		0://等待激活
			IF   xcmd THEN
			 		xQBusy:=TRUE;
					xQDone:=FALSE;
					iCmdStep :=iCmdStep +1;
					xcmd:=FALSE;
			END_IF
		1://指令
				iCmdStep :=iCmdStep +1;
				iCmdOldStep:=iCmdStep;
		2://开始执行
				xStart :=TRUE;
				iCmdStep :=iCmdStep +1;
				iCmdOldStep:=iCmdStep;
		3://等待接受
					IF   xBusy THEN
					 		iCmdStep :=iCmdStep +1;
					END_IF
					iCmdOldStep:=iCmdStep;
		4://报警待整理数据
				IF  iOperType<> 14  AND  NOT xBusy AND xDone THEN
						iCmdStep :=iCmdStep +1;
				ELSIF iOperType =14 AND  NOT xQNoRead THEN
				 		iCmdStep :=iCmdStep +1;	
				END_IF
				iCmdOldStep:=iCmdStep;
		5://处理接收的数据
					IF iOperType =1 THEN
							IF FIND(strQBarCode,'$R') <> 0 AND FIND(strQBarCode,'I4') <> 0	THEN					
									 CutStrToSeperator('"',strQBarCode);
									 stParOut.sSrialNumber := CutStrToSeperator('"',strQBarCode);
									 iCmdStep :=iCmdStep +1;;	
							END_IF
					ELSIF iOperType =2 THEN
					 					IF FIND(strQBarCode,'$R') <> 0 		THEN
															IF FIND(strQBarCode,'S') <> 0 THEN
																			_Stemp[1]:=RIGHT(strQBarCode,LEN(strQBarCode)-4);
																			_Stemp[2]:=LEFT(_Stemp[1],FIND(_Stemp[1],'g$R')-1);
																			stParOut.rCurrentTareWight := TO_REAL(_Stemp[2]);
																			iCmdStep :=iCmdStep +1;	
															ELSIF FIND(strQBarCode,'T +') <> 0 THEN	
																			eErrorID:=MT_MCK_ERROR.FLT_ZOverMax;
															ELSIF FIND(strQBarCode,'T -') <> 0 THEN	
																			eErrorID:=MT_MCK_ERROR.FLT_ZOverMax;
															ELSIF FIND(strQBarCode,'T I') <> 0 THEN
															 				eErrorID:=MT_MCK_ERROR.FLT_CannotExecutable;			
															END_IF										
									END_IF						
					ELSIF iOperType =3 THEN
					 						IF FIND(strQBarCode,'$R') <> 0 		THEN
															IF FIND(strQBarCode,'TI S') <> 0 OR FIND(strQBarCode,'TI D') <> 0 THEN
																_Stemp[1]:=RIGHT(strQBarCode,LEN(strQBarCode)-4);
																_Stemp[2]:=LEFT(_Stemp[1],FIND(_Stemp[1],'g$R')-1);
																stParOut.rCurrentTareWight := TO_REAL(_Stemp[2]);
																iCmdStep :=iCmdStep +1;;	
															ELSIF FIND(strQBarCode,'TI +') <> 0 THEN	
																eErrorID:=MT_MCK_ERROR.FLT_ZOverMax;
															ELSIF FIND(strQBarCode,'TI -') <> 0 THEN	
																eErrorID:=MT_MCK_ERROR.FLT_ZOverMax;
															ELSIF FIND(strQBarCode,'TI I') <> 0 THEN
															  eErrorID:=MT_MCK_ERROR.FLT_CannotExecutable;			
															END_IF										
												END_IF		
					ELSIF iOperType =4 THEN									
										IF FIND(strQBarCode,'$R') <> 0 AND FIND(strQBarCode,'TA') <> 0	THEN
											 _Stemp[1]:=RIGHT(strQBarCode,LEN(strQBarCode)-5);
											 _Stemp[2]:=LEFT(_Stemp[1],FIND(_Stemp[1],'g$R')-1);
											 stParOut.rCurrentTareWight := TO_REAL(_Stemp[2]);
											 iCmdStep :=iCmdStep +1;;	
										END_IF		
					ELSIF	iOperType =5 THEN		
										IF FIND(strQBarCode,'$R') <> 0 AND FIND(strQBarCode,'TAC') <> 0	THEN
											 stParOut.rCurrentTareWight:=0;
											 iCmdStep :=iCmdStep +1;;	
										 ELSIF FIND(strQBarCode,'EL') <>0 THEN
											 eErrorID:=MT_MCK_ERROR.FLT_LogicaL;//逻辑错误
										 ELSIF FIND(strQBarCode,'ES') <>0 THEN
											 eErrorID:=MT_MCK_ERROR.FLT_Syntax;//语法错误
										 ELSIF FIND(strQBarCode,'I') <>0 THEN
											 eErrorID:=MT_MCK_ERROR.FLT_CommandCantSend;//指令条件不满足,无法发送	
										 ELSIF FIND(strQBarCode,'L') <>0 THEN
											 eErrorID:=MT_MCK_ERROR.FLT_PARA;//参数错误		
										 ELSIF FIND(strQBarCode,'TAC I') <>0 THEN
											 eErrorID:=MT_MCK_ERROR.FLT_CommandCantSend;
										 END_IF																	
					ELSIF  	iOperType =6 THEN													
											IF FIND(strQBarCode,'Z A') <> 0 THEN
													stParOut.rCurrentTareWight :=0;
													stParOut.rCurrentWeight :=0;
													iCmdStep :=iCmdStep +1;;	
											ELSIF FIND(strQBarCode,'Z +') <> 0 THEN
												eErrorID:=MT_MCK_ERROR.FLT_ZOverMax;							
											ELSIF FIND(strQBarCode,'Z -') <> 0 THEN
												eErrorID:=MT_MCK_ERROR.FLT_ZOverMin;				
											ELSIF FIND(strQBarCode,'Z I') <> 0 THEN
												eErrorID:=MT_MCK_ERROR.FLT_CannotExecutable;					
											END_IF			
				ELSIF  	iOperType =7 THEN													
											IF FIND(strQBarCode,'$R') <> 0 	THEN
														 IF FIND(strQBarCode,'ZI') <> 0 AND (FIND(strQBarCode,'S') <> 0 OR FIND(strQBarCode,'D') <> 0) THEN
															 stParOut.rCurrentTareWight :=0;
															 stParOut.rCurrentWeight :=0;
															 iCmdStep :=iCmdStep +1;;	
															ELSIF FIND(strQBarCode,'Z +') <> 0 THEN
																	 eErrorID:=MT_MCK_ERROR.FLT_ZOverMax;							
															 ELSIF FIND(strQBarCode,'Z -') <> 0 THEN
																	 eErrorID:=MT_MCK_ERROR.FLT_ZOverMin;				
																ELSIF FIND(strQBarCode,'Z I') <> 0 THEN
																	 eErrorID:=MT_MCK_ERROR.FLT_ZI;		
																ELSIF	 FIND(strQBarCode,'ZI I') <> 0 THEN
																 	 eErrorID:=MT_MCK_ERROR.FLT_CannotExecutable;
																END_IF
													END_IF
					ELSIF  	iOperType =8 THEN												
											IF FIND(strQBarCode,'$R') <> 0 AND FIND(strQBarCode,'S') <>0		THEN
														IF FIND(strQBarCode,'mg') <> 0 THEN
															_Stemp[1]:=RIGHT(strQBarCode,LEN(strQBarCode)-5);
															_Stemp[2]:=LEFT(_Stemp[1],FIND(_Stemp[1],'g$R')-1);
															stParOut.rCurrentWeight := TO_REAL(_Stemp[2]);
															stParOut.sWeightUnit:='mg';
															iCmdStep :=iCmdStep +1;;	
														ELSE 
															IF FIND(strQBarCode,'g') <> 0 THEN
																_Stemp[1]:=RIGHT(strQBarCode,LEN(strQBarCode)-5);
																_Stemp[2]:=LEFT(_Stemp[1],FIND(_Stemp[1],'g$R')-1);
																stParOut.rCurrentWeight := TO_REAL(_Stemp[2]);
																stParOut.sWeightUnit:='mg';		
																iCmdStep :=iCmdStep +1;;			
															END_IF				
														END_IF
											ELSIF FIND(strQBarCode,'EL') <>0 THEN
														eErrorID:=MT_MCK_ERROR.FLT_LogicaL;//逻辑错误
											ELSIF FIND(strQBarCode,'ES') <>0 THEN
														eErrorID:=MT_MCK_ERROR.FLT_Syntax;//语法错误		
										ELSIF FIND(strQBarCode,'I') <>0 THEN
														eErrorID:=MT_MCK_ERROR.FLT_CommandCantSend;//指令条件不满足,无法发送		
										ELSIF FIND(strQBarCode,'L') <>0 THEN
														eErrorID:=MT_MCK_ERROR.FLT_PARA;//参数错误	
										ELSIF FIND(strQBarCode,'S I') <>0 THEN
											 eErrorID:=MT_MCK_ERROR.FLT_CannotExecutable;
										END_IF			
					ELSIF  	iOperType =9 THEN							
										IF FIND(strQBarCode,'$R') <> 0 AND FIND(strQBarCode,'S') <>0 THEN
													 IF FIND(strQBarCode,'g') <> 0 THEN
														 _Stemp[1]:=RIGHT(strQBarCode,LEN(strQBarCode)-5);
														 _Stemp[2]:=LEFT(_Stemp[1],FIND(_Stemp[1],'g$R')-1);
														 stParOut.rCurrentWeight := TO_REAL(_Stemp[2]);
														 stParOut.sWeightUnit:='mg';	
															iCmdStep :=iCmdStep +1;;				
													 ELSE 
														 IF FIND(strQBarCode,'g') <> 0 THEN
															 _Stemp[1]:=RIGHT(strQBarCode,LEN(strQBarCode)-5);
															 _Stemp[2]:=LEFT(_Stemp[1],FIND(_Stemp[1],'g$R')-1);
															 stParOut.rCurrentWeight := TO_REAL(_Stemp[2]);
															 stParOut.sWeightUnit:='mg';		
																iCmdStep :=iCmdStep +1;;			
														 END_IF				
													 END_IF
													 IF stParOut.rCurrentWeight>stParOut.rWeightMax THEN
														 stParOut.rWeightMax:=stParOut.rCurrentWeight;
													 END_IF
													 IF stParOut.rCurrentWeight<stParOut.rWeightMin THEN
														 stParOut.rWeightMin:=stParOut.rCurrentWeight;
													 END_IF	
													
										ELSIF FIND(strQBarCode,'EL') <>0 THEN
													 eErrorID:=MT_MCK_ERROR.FLT_LogicaL;//逻辑错误
													
										ELSIF FIND(strQBarCode,'ES') <>0 THEN
													 eErrorID:=MT_MCK_ERROR.FLT_Syntax;//语法错误
																
										 ELSIF FIND(strQBarCode,'I') <>0 THEN
													 eErrorID:=MT_MCK_ERROR.FLT_CommandCantSend;//指令条件不满足,无法发送
																	
										ELSIF FIND(strQBarCode,'L') <>0 THEN
													 eErrorID:=MT_MCK_ERROR.FLT_PARA;//参数错误
										ELSIF FIND(strQBarCode,'SI I') <>0 THEN
											 eErrorID:=MT_MCK_ERROR.FLT_CannotExecutable;//无法执行		
										END_IF		
				ELSIF  	iOperType =10 THEN										
												IF FIND(strQBarCode,'$R') <> 0 AND FIND(strQBarCode,'S') <>0				THEN
													 IF FIND(strQBarCode,'g') <> 0 THEN
														 _Stemp[1]:=RIGHT(strQBarCode,LEN(strQBarCode)-5);
														 _Stemp[2]:=LEFT(_Stemp[1],FIND(_Stemp[1],'g$R')-1);
														 stParOut.rCurrentWeight := TO_REAL(_Stemp[2]);
														 stParOut.sWeightUnit:='mg';
														 iCmdStep :=iCmdStep +1;;	
													 ELSE 
														 IF FIND(strQBarCode,'g') <> 0 THEN
															 _Stemp[1]:=RIGHT(strQBarCode,LEN(strQBarCode)-5);
															 _Stemp[2]:=LEFT(_Stemp[1],FIND(_Stemp[1],'g$R')-1);
															 stParOut.rCurrentWeight := TO_REAL(_Stemp[2]);
															 stParOut.sWeightUnit:='mg';	
																iCmdStep :=iCmdStep +1;;				
														 END_IF				
													 END_IF
										 ELSIF FIND(strQBarCode,'EL') <>0 THEN
											 eErrorID:=MT_MCK_ERROR.FLT_LogicaL;//逻辑错误
										 ELSIF FIND(strQBarCode,'ES') <>0 THEN
											 eErrorID:=MT_MCK_ERROR.FLT_Syntax;//语法错误				
										 ELSIF FIND(strQBarCode,'I') <>0 THEN
											 eErrorID:=MT_MCK_ERROR.FLT_CommandCantSend;//指令条件不满足,无法发送 			
										 ELSIF FIND(strQBarCode,'L') <>0 THEN
											 eErrorID:=MT_MCK_ERROR.FLT_PARA;//参数错误
										 ELSIF FIND(strQBarCode,'SIR I') <>0 THEN
											 eErrorID:=MT_MCK_ERROR.FLT_CannotExecutable;//无法执行
										END_IF
				ELSIF  	iOperType =11 THEN										 
									IF FIND(strQBarCode,'$R') <> 0 AND FIND(strQBarCode,'S') <> 0		THEN
												 _Stemp[1]:=RIGHT(strQBarCode,LEN(strQBarCode)-4);
											_Stemp[2]:=LEFT(_Stemp[1],FIND(_Stemp[1],'g$R')-1);
											stParOut.rCurrentWeight := TO_REAL(_Stemp[2]);
											iCmdStep :=iCmdStep +1;;	
									END_IF														 
				ELSIF  	iOperType =12 THEN						
					 				IF FIND(strQBarCode,'$R') <> 0 AND FIND(strQBarCode,'I4') <> 0	THEN
										CutStrToSeperator('"',strQBarCode);
										stParOut.sSrialNumber := CutStrToSeperator('"',strQBarCode);
										iCmdStep :=iCmdStep +1;	
									END_IF
				ELSIF  	iOperType =13 THEN			
								IF FIND(strQBarCode,'$R') <> 0 AND FIND(strQBarCode,'I4') <> 0	THEN
												iCmdStep :=iCmdStep +1;	
								ELSE			
								 					iCmdStep :=2;	
								END_IF
				ELSIF   iOperType =14 THEN	
							  IF FIND(strQBarCode,'$R') <> 0 AND FIND(strQBarCode,'S S') <> 0	THEN
									//稳态
								 				IF    FIND(strQBarCode,'g')<>0 THEN
												   // stParOut.rRepeatWeight:=strQBarCode;
													//	stParOut.rStableWeight:=strQBarCode;
													_Stemp[1]:=RIGHT(strQBarCode,LEN(strQBarCode)-5);
													_Stemp[2]:=LEFT(_Stemp[1],FIND(_Stemp[1],'g$R')-1);
													stParOut.rRepeatWeight:=TO_REAL(_Stemp[2]);
													stParOut.rStableWeight:=stParOut.rRepeatWeight;
													xRepeatReceive:=TRUE;;
												ELSE
												 			eErrorID:=MT_MCK_ERROR.FLT_SIRERROR;
												 END_IF
												iCmdStep :=iCmdStep +1;	
								ELSIF  	FIND(strQBarCode,'$R') <> 0 AND FIND(strQBarCode,'S D')<>0 THEN
								 //非稳态
								 					IF    FIND(strQBarCode,'g')<>0 THEN
																_Stemp[1]:=RIGHT(strQBarCode,LEN(strQBarCode)-5);
																_Stemp[2]:=LEFT(_Stemp[1],FIND(_Stemp[1],'g$R')-1);
																stParOut.rRepeatWeight:=TO_REAL(_Stemp[2]);
													 			xRepeatReceive:=TRUE;
													ELSE
												 			eErrorID:=MT_MCK_ERROR.FLT_SIRERROR;
												 END_IF
												iCmdStep :=iCmdStep +1;	
								ELSIF  FIND(strQBarCode,'S I')<>0 THEN
								 			eErrorID:=MT_MCK_ERROR.FLT_CannotExecutable;//无法执行
								ELSIF  FIND(strQBarCode,'S L')<>0 THEN
								 			eErrorID:=MT_MCK_ERROR.FLT_PARA;//参数错误
								ELSIF  FIND(strQBarCode,'S +')<>0 THEN
								 			eErrorID:=MT_MCK_ERROR.FLT_SIROverMax;
								ELSIF  FIND(strQBarCode,'S -')<>0 THEN
								 			eErrorID:=MT_MCK_ERROR.FLT_SIROverMIN;
								END_IF				
				END_IF
				iCmdOldStep:=iCmdStep;
		6:	
						xQDone:=TRUE;
						xQBusy:=FALSE;	
						iCmdOldStep:=iCmdStep;
						iCmdStep :=0;		
	END_CASE
END_ACTION

ACTION ACT_Error:
IF  eErrorID <> 0 THEN
	xQError:=TRUE;
END_IF
//报错内容输出
CASE eErrorID OF 
	MT_MCK_ERROR.FLT_CMD_TIMEOUT:
		stParOut.sErrorID:='FLT_CMD_TIMEOUT';
	MT_MCK_ERROR.FLT_CmdFeedback:
		stParOut.sErrorID:='FLT_CmdFeedback';
	MT_MCK_ERROR.FLT_CommandCantSend:
		stParOut.sErrorID:='FLT_CommandCantSend';
	MT_MCK_ERROR.FLT_CONNECT:
		stParOut.sErrorID:='FLT_CONNECT';
	MT_MCK_ERROR.FLT_LogicaL:
		stParOut.sErrorID:='FLT_LogicaL';
	MT_MCK_ERROR.FLT_Par:
		stParOut.sErrorID:='FLT_Par';
	MT_MCK_ERROR.FLT_PARA:
		stParOut.sErrorID:='FLT_PARA';
	MT_MCK_ERROR.FLT_RDYCMD:
		stParOut.sErrorID:='FLT_RDYCMD';
	MT_MCK_ERROR.FLT_STOP_TIMEOUT:
		stParOut.sErrorID:='FLT_STOP_TIMEOUT';
	MT_MCK_ERROR.FLT_Syntax:
		stParOut.sErrorID:='FLT_Syntax';
	MT_MCK_ERROR.FLT_TOverMax:
		stParOut.sErrorID:='FLT_TOverMax';
	MT_MCK_ERROR.FLT_TOverMin:
		stParOut.sErrorID:='FLT_TOverMin';
	MT_MCK_ERROR.FLT_ZI:
		stParOut.sErrorID:='FLT_ZI';
	MT_MCK_ERROR.FLT_ZOverMax:
		stParOut.sErrorID:='FLT_ZOverMax';
	MT_MCK_ERROR.FLT_ZOverMin:
		stParOut.sErrorID:='FLT_ZOverMin';
	MT_MCK_ERROR.FLT_CannotExecutable:
			stParOut.sErrorID:='FLT_CannotExecutable';	
	MT_MCK_ERROR.No_ERROR:
		stParOut.sErrorID:='No_ERROR';		
END_CASE
END_ACTION

ACTION ACT_OP:
OperR_TRIG[1](CLK:= (xManualMode AND  stDeviceOpe.xReadSerialNum_HMI) OR((xAutoMode OR  xIDeviceRunning) AND stDeviceOpe.xReadSerialNum_Auto) , Q=> );	//获取序列号,I4			
OperR_TRIG[2](CLK:= (xManualMode AND  stDeviceOpe.xShelling_HMI) OR((xAutoMode OR  xIDeviceRunning) AND stDeviceOpe.xShelling_Auto) , Q=> );		//稳态去皮重,T		
OperR_TRIG[3](CLK:= (xManualMode AND  stDeviceOpe.xShellingInstanly_HMI) OR((xAutoMode OR  xIDeviceRunning) AND stDeviceOpe.xShellingInstanly_HMI) , Q=> );	//立即去皮重,TI			
OperR_TRIG[4](CLK:= (xManualMode AND  stDeviceOpe.xSetTare_HMI) OR((xAutoMode OR  xIDeviceRunning) AND stDeviceOpe.xSetTare_Auto) , Q=> );		//预置皮重，TA		
OperR_TRIG[5](CLK:= (xManualMode AND  stDeviceOpe.xlearTare_HMI) OR((xAutoMode OR  xIDeviceRunning) AND stDeviceOpe.xlearTare_Auto) , Q=> );	//清除皮重,TAC			
OperR_TRIG[6](CLK:= (xManualMode AND  stDeviceOpe.xClearZero_HMI) OR((xAutoMode OR  xIDeviceRunning) AND stDeviceOpe.xClearZero_Auto) , Q=> );	//稳态清零,Z	
OperR_TRIG[7](CLK:= (xManualMode AND  stDeviceOpe.xClearZeroInstanly_HMI) OR((xAutoMode OR  xIDeviceRunning) AND stDeviceOpe.xClearZeroInstanly_Auto) , Q=> );	////立即清零,ZI	
OperR_TRIG[8](CLK:= (xManualMode AND  stDeviceOpe.xAcquireWeight_Steady_HMI) OR((xAutoMode OR  xIDeviceRunning) AND stDeviceOpe.xClearZero_Auto) , Q=> );	////单次获取稳态重量,S	
OperR_TRIG[9](CLK:= (xManualMode AND  stDeviceOpe.xAcquireWeight_RealTime_HMI) OR((xAutoMode OR  xIDeviceRunning) AND stDeviceOpe.xAcquireWeight_RealTime_Auto) , Q=> );	////连续获取重量,SI
OperR_TRIG[10](CLK:= (xManualMode AND  stDeviceOpe.xAcquireWeight_Continuous_HMI) OR((xAutoMode OR  xIDeviceRunning) AND stDeviceOpe.xAcquireWeight_Continuous_Auto) , Q=> );	////连续获取重量,SIR	
OperR_TRIG[11](CLK:= (xManualMode AND  stDeviceOpe.xAcquireWeight_Stop_HMI) OR((xAutoMode OR  xIDeviceRunning) AND stDeviceOpe.xAcquireWeight_Stop_Auto) , Q=> );	///中断连续获取重量,SI
OperR_TRIG[12](CLK:= (xManualMode AND  stDeviceOpe.xRestart_HMI) OR((xAutoMode OR  xIDeviceRunning) AND stDeviceOpe.xRestart_Auto) , Q=> );	//重启秤体	
OperR_TRIG[13](CLK:=xIReset , Q=> );	//Cancel	
OperR_TRIG[14](CLK:=( (xManualMode AND  stDeviceOpe.xRepeatRead_Hmi ) OR((xAutoMode OR  xIDeviceRunning) AND stDeviceOpe.xRepeatRead_Auto) )AND iOperType <>14 , Q=> );	//循环读取重量并显示
FOR  i:= 1 TO 20 BY 1 DO
 	IF   OperR_TRIG[i].Q THEN
				iOperType:= i;
				xCmd:=TRUE;
				EXIT;
	END_IF
END_FOR

IF   iOperType =1 THEN
 	strRead := 'I4$R$N';
ELSIF   iOperType =2 THEN
 	strRead := 'T$R$N';
ELSIF   iOperType =3 THEN
 	strRead := 'TI$R$N';
ELSIF   iOperType =4 THEN
 	_sSendData := CONCAT(_sSendData,'TA');
	_sSendData := CONCAT(_sSendData,' ');		
	_sSendData := CONCAT(_sSendData,TO_STRING(rTareSet));
	_sSendData := CONCAT(_sSendData,' ');
	_sSendData := CONCAT(_sSendData,'g');//单位
	_sSendData := CONCAT(_sSendData,'$R$N');//回车换行符			
 	strRead := _sSendData;
ELSIF   iOperType =5 THEN
 	strRead := 'TAC$R$N';
ELSIF   iOperType =6 THEN
 	strRead := 'Z$R$N';
ELSIF   iOperType =7 THEN
 	strRead := 'ZI$R$N';
ELSIF   iOperType =8 THEN
 	strRead := 'S$R$N';
ELSIF   iOperType =9 THEN
 	strRead := 'SI$R$N';
ELSIF   iOperType =10 THEN
 	strRead := 'SIR$R$N';
ELSIF   iOperType =11 THEN
 	strRead := 'SI$R$N';
ELSIF   iOperType =12 THEN
 	strRead := 'R01$R$N';
ELSIF iOperType =13 THEN
 	strRead := '@$R$N';
ELSIF  iOperType =14 THEN
  strRead := 'SIR$R$N';
END_IF

	stDeviceOpe.xReadSerialNum_HMI:=stDeviceOpe.xReadSerialNum_Auto :=FALSE;	//获取序列号,I4
	stDeviceOpe.xShelling_HMI:=stDeviceOpe.xShelling_Auto						:=FALSE;//稳态去皮重,T
	stDeviceOpe.xShellingInstanly_HMI:=stDeviceOpe.xShellingInstanly_Auto	:=FALSE;//立即去皮重,TI	
	stDeviceOpe.xSetTare_HMI:=stDeviceOpe.xSetTare_Auto										:=FALSE;//预置皮重，TA
	stDeviceOpe.xlearTare_HMI:=stDeviceOpe.xlearTare_Auto									:=FALSE;//清除皮重,TAC
	stDeviceOpe.xClearZero_HMI:=stDeviceOpe.xClearZero_Auto								:=FALSE;//稳态清零,Z
	stDeviceOpe.xClearZeroInstanly_HMI:=stDeviceOpe.xClearZeroInstanly_Auto:=FALSE;//立即清零,ZI
	stDeviceOpe.xAcquireWeight_Steady_HMI:=stDeviceOpe.xAcquireWeight_Steady_Auto :=FALSE;//单次获取稳态重量,S
	stDeviceOpe.xAcquireWeight_RealTime_HMI:=stDeviceOpe.xAcquireWeight_RealTime_Auto:=FALSE;//连续获取重量,SI
	stDeviceOpe.xAcquireWeight_Continuous_HMI:=stDeviceOpe.xAcquireWeight_Continuous_Auto:=FALSE;//连续获取重量,SIR
	stDeviceOpe.xAcquireWeight_Stop_HMI:=stDeviceOpe.xAcquireWeight_Stop_Auto		:=FALSE;//中断连续获取重量,SI
	stDeviceOpe.xRestart_HMI:=stDeviceOpe.xRestart_Auto										      :=FALSE;//重启秤体	
	stDeviceOpe.xRepeatRead_Hmi:=stDeviceOpe.xRepeatRead_Auto							      :=FALSE;//重复读取
	//xIReset:=FALSE;
END_ACTION

ACTION ACT_Reset:
IF ( xIReset = TRUE )THEN
 		iCmdStep:=0;
  	iStep := 0 ;
		iLoadStep:=0;
  	xQError := FALSE ;
  	xBusy  := FALSE;
		xQBusy  := FALSE;
		xStart  := FALSE;
		eErrorID:=MT_MCK_ERROR.No_ERROR;
		iCmdOldStep:=0;
		xIReset:=FALSE;
END_IF
END_ACTION

ACTION ACT_RW:

 
IF ( First = FALSE )THEN
   	TcpIpClient.sRemoteServer := stSysPar.sRemoteHost;
 		TcpIpClient.nRemotePort := stSysPar.nRemotePort;
   	TcpIpClient.pSendData := ADR(ClientSendBuffer);
   	TcpIpClient.pRecvData := ADR(ClientRecvBuffer);
   	First := TRUE ;
ELSE
  	TcpIpClient(iStep :=	eStepCmd );
 	CASE iStep OF
		0: (* wait start *)
		   	IF ( xStart = FALSE )THEN
		       	xDone := FALSE ;
		   	END_IF
		  	IF ( xStart = FALSE ) AND( xDone = FALSE )THEN
		       	xRdyCmd := TRUE  ;
		   	END_IF

		   	IF ( xStart = TRUE ) AND( xRdyCmd = TRUE )THEN
				iStep  :=  10 ;
				xBusy:=TRUE;
			  xRdyCmd := FALSE  ;
			(*ELSE
 			 	xBusy  := FALSE;*)
		   	END_IF

		10: (* creat soket*)
			xStart := FALSE;
			MEMSET(ADR(strLocalQBarCode),0,SIZEOF(strLocalQBarCode));
			MEMSET(ADR(strQBarCode),0,SIZEOF(strQBarCode));
			MEMSET(ADR(ClientRecvBuffer),0,SIZEOF(ClientRecvBuffer));
			eStepCmd := CLIENT_STATE_CONNECT_START ;
		    	iStep := 20 ;

		20: (* socket ok *)
 			 IF( eStepCmd = CLIENT_STATE_IDLE )THEN
		    	 	iStep := 30 ;
			ELSIF( eStepCmd = CLIENT_STATE_ERROR )THEN
				iQErrorNo:=iStep;
		    	 	iStep := 100 ;
	         	END_IF

		30: (* send read *)
   			MEMCPY(ADR(ClientSendBuffer),ADR(strRead),SIZEOF(strRead));
			TcpIpClient.SendLen := LEN(strRead);
			eStepCmd := CLIENT_STATE_SEND_START ;
		    	iStep := 40 ;

		40: (* send ok *)
 			IF( eStepCmd = CLIENT_STATE_IDLE )THEN
		    	 	iStep := 50 ;
			ELSIF( eStepCmd = CLIENT_STATE_ERROR )THEN
				iQErrorNo:=iStep;
		    	 	iStep := 999 ;
	         	END_IF

		50: (* recive read *)
			xQNoRead:=TRUE;
			eStepCmd := CLIENT_STATE_RECIVE_START ;
		    	iStep := 55 ;

   55:
			strLocalQBarCode:='';
			strQBarCode:='';
			Waittime(IN:=TRUE, PT:= t#20ms);
	      	IF(waittime.Q = TRUE )THEN
 							Waittime(IN:= FALSE);
		    	 		iStep := 60 ;
	        END_IF

		60: (* recive end *)
				IF( eStepCmd = CLIENT_STATE_IDLE )THEN
						 MEMCPY(ADR(strLocalQBarCode),ADR(ClientRecvBuffer),TcpIpClient.cbReceived);
						 strQBarCode:=MID(strLocalQBarCode,iICodeLEN,iICodePOS);
						 iStep := 80 ;
			 ELSIF( eStepCmd = CLIENT_STATE_ERROR )THEN
				 		 iQErrorNo:=iStep;
						 iStep := 70;
			 END_IF
		70:
				MEMSET(ADR(strLocalQBarCode),0,SIZEOF(strLocalQBarCode));
				MEMSET(ADR(strQBarCode),0,SIZEOF(strQBarCode));
				iStep := 80;

		80: (* close socket *)
			 IF  strQBarCode<>'' THEN
							 xQNoRead:=FALSE;
			 ELSE
							 xQNoRead:=TRUE;
			 END_IF
			 IF iOperType =14 THEN
					 	iStep := 50 ;
			 ELSE
				 		iStep := 100 ;
			 END_IF
		100: (* close socket *)
					eStepCmd := CLIENT_STATE_CLOSE_START ;
		    	iStep := 110 ;
		110: (* recive end *)
				IF( eStepCmd = CLIENT_STATE_IDLE )THEN
							xBusy  := FALSE;
							xDone := TRUE ;
							iStep := 0 ;
				ELSIF( eStepCmd = CLIENT_STATE_ERROR )THEN
							iStep := 999 ;
							END_IF

		999: (* Done *)
				 xBusy:=FALSE;
				 xQError := TRUE ;
					iStep := 0 ;
	END_CASE
END_IF
END_ACTION

END_FUNCTION_BLOCK

// ---- POUs/003_FB/0008_LocalClient/FB_LocalClient.TcPOU
FUNCTION_BLOCK FB_LocalClient
VAR_INPUT
	sRemoteServer		: STRING(15) := '192.168.0.3';(* IP adress of remote server *)
	nRemotePort			: UDINT := 1030;
    RecvTime            : TIME ;
	pSendData           : POINTER TO BYTE ;
    SendLen             : INT ;
	pRecvData           : POINTER TO BYTE ;
    RecvLen             : INT := 255 ;


    Start             : BOOL ;
    Send              : BOOL ;
    Recv              : BOOL ;
    Close             : BOOL ;

END_VAR
VAR_OUTPUT
			hSocket				: T_HSOCKET;
			bBusy 				: BOOL;
			bError				: BOOL;
			nErrId				: UDINT;
    Connected           : BOOL ;
    SendOK              : BOOL ;
    RecvOK              : BOOL ;
    Closed              : BOOL ;
    RdyCmd              : BOOL ;
	Done: BOOL;
END_VAR

VAR_IN_OUT
    iStep             : E_ClientSteps;
END_VAR


VAR
	
	
	fbConnect 		: FB_SocketConnect := ( sSrvNetId := ''  );
	fbClose				: FB_SocketClose := ( sSrvNetId := '', tTimeout := DEFAULT_ADS_TIMEOUT );
	fbSocketSend		: FB_SocketSend      := ( sSrvNetID := '', tTimeout := DEFAULT_ADS_TIMEOUT );
	fbSocketReceive        : FB_SocketReceive := ( sSrvNetID := '', tTimeout := DEFAULT_ADS_TIMEOUT );
	fbConnectTON		: TON := ( PT := PLCPRJ_RECONNECT_TIME );
	fbDataExchaTON		: TON := ( PT := PLCPRJ_SEND_CYCLE_TIME );
	fbReceiveTON		: TON;
	fbDisconnectTON      : TON;
    arrayRecive                 : ARRAY [1..1000] OF BYTE ;
	a,b,c,d : BOOL ;

	cbReceived, startPos, endPos, idx	: UDINT;
	cbFrame				: UDINT;
	rxBuffer				: ARRAY[0..MAX_PLCPRJ_RXBUFFER_SIZE] OF BYTE;
	
END_VAR

CASE iStep OF
	CLIENT_STATE_IDLE:
	;
	CLIENT_STATE_CONNECT_START:
		  IF ( Connected =  FALSE )
		  THEN
				fbConnectTON( IN := TRUE, PT := PLCPRJ_RECONNECT_TIME );
						IF fbConnectTON.Q THEN
							fbConnectTON( IN := FALSE );
							fbConnect(  bExecute := FALSE  );
							fbConnect(	sRemoteHost		:= sRemoteServer,
										nRemotePort		:= nRemotePort,
										bExecute		:= TRUE );
							iStep := CLIENT_STATE_CONNECT_WAIT;
						END_IF

	    	ELSE
			   iStep := CLIENT_STATE_IDLE;
			END_IF

   CLIENT_STATE_CONNECT_WAIT:
				fbConnect( bExecute := FALSE );
				IF NOT fbConnect.bBusy THEN
					IF NOT fbConnect.bError THEN
						Connected 	:= TRUE;
						hSocket 	:= fbConnect.hSocket;
						iStep := CLIENT_STATE_IDLE;

					ELSE

						nErrId := fbConnect.nErrId;
						iStep := CLIENT_STATE_ERROR;
					END_IF
				END_IF


	CLIENT_STATE_SEND_START:
		fbSocketSend( bExecute := FALSE );
		fbSocketSend( 	hSocket	:= hSocket,
						pSrc	:= pSendData,
						cbLen	:= SendLen,(* string length inclusive zero delimiter *)
						bExecute:= TRUE );
		cbReceived	:= 0 ;
		MEMSET(ADR(rxBuffer),0,SIZEOF(rxBuffer));
		iStep := CLIENT_STATE_SEND_WAIT;

	CLIENT_STATE_SEND_WAIT:
		fbSocketSend( bExecute := FALSE );
		IF NOT fbSocketSend.bBusy THEN
			IF NOT fbSocketSend.bError THEN
				iStep := CLIENT_STATE_IDLE;
			ELSE

				nErrId := fbSocketSend.nErrId;
				iStep := CLIENT_STATE_CLOSE_START;
			END_IF
		END_IF
	CLIENT_STATE_WAITTIME1:
		iStep := CLIENT_STATE_WAITTIME2;
	CLIENT_STATE_WAITTIME2:
		iStep := CLIENT_STATE_RECIVE_START;

	CLIENT_STATE_RECIVE_START:
		fbDisconnectTON(  );
		fbReceiveTON( IN := TRUE );
		IF fbReceiveTON.Q THEN
			fbReceiveTON( IN := FALSE );
			fbSocketReceive( bExecute := FALSE );
			fbSocketReceive(  hSocket:= hSocket,
							pDest:= ADR( rxBuffer ) + cbReceived,
							cbLen:= SIZEOF( rxBuffer ) - cbReceived,
							bExecute:= TRUE );
			iStep := CLIENT_STATE_RECIVE_WAIT;
		END_IF

	CLIENT_STATE_RECIVE_WAIT:
		fbSocketReceive( bExecute := FALSE );
		IF NOT fbSocketReceive.bBusy THEN
			IF NOT fbSocketReceive.bError THEN

				IF (fbSocketReceive.nRecBytes > 0) THEN(* bytes received *)

					startPos 		:= cbReceived;(* rxBuffer array index of first data byte *)
					endPos  		:= cbReceived + fbSocketReceive.nRecBytes  - 1;(* rxBuffer array index of last data byte *)
					cbReceived 	:= cbReceived + fbSocketReceive.nRecBytes;(* calculate the number of received data bytes *)
					cbFrame		:= 0;(* reset frame length *)

					IF cbReceived < RecvLen THEN(* no overflow *)

						fbReceiveTON( PT := T#0s ); (* bytes received => increase the read (polling) speed *)
						fbDisconnectTON( IN := FALSE );(* bytes received => disable timeout check *)

						(* search for string end delimiter *)
						FOR idx := startPos TO endPos BY 1 DO
							IF rxBuffer[idx] = 0 THEN(* string end delimiter found *)
								cbFrame := idx + 1;(* calculate the length of the received string (inclusive the end delimiter) *)
								MEMCPY(  pRecvData, ADR( rxBuffer ), cbFrame );(* copy the received string to the output variable (inclusive the end delimiter) *)
								MEMMOVE( ADR( rxBuffer ), ADR( rxBuffer[cbFrame] ),  cbReceived - cbFrame  );(* move the reamaining data bytes *)
								cbReceived := cbReceived - cbFrame;(* recalculate the reamaining data byte length *)
								a := TRUE ;
								iStep := CLIENT_STATE_IDLE;
								EXIT;
							END_IF
						END_FOR

					ELSE(* there is no more free read buffer space => the answer string should be terminated *)
						b := TRUE ;
						nErrId := PLCPRJ_ERROR_RECEIVE_BUFFER_OVERFLOW;(* buffer overflow !*)
						iStep := CLIENT_STATE_CLOSE_START;
					END_IF

				ELSE(* no bytes received *)
					fbReceiveTON( PT := PLCPRJ_RECEIVE_POLLING_TIME );(* no bytes received => decrease the read (polling) speed *)
					fbDisconnectTON( IN := TRUE, PT := PLCPRJ_RECEIVE_TIMEOUT );(* no bytes received => enable timeout check*)
					IF fbDisconnectTON.Q THEN (* timeout error*)
						fbDisconnectTON( IN := FALSE );
						c := TRUE ;
						nErrID := PLCPRJ_ERROR_RECEIVE_TIMEOUT;
						iStep := CLIENT_STATE_IDLE;
					ELSE(* repeat reading *)
						iStep := CLIENT_STATE_RECIVE_START; (* repeat reading *)
					END_IF
				END_IF
			ELSE(* receive error *)
				d := TRUE ;
				nErrId := fbSocketReceive.nErrId;
				iStep := CLIENT_STATE_CLOSE_START;
			END_IF
		END_IF



	CLIENT_STATE_CLOSE_START:
	    fbClose( bExecute := FALSE );
		fbClose(	hSocket:= hSocket,
				bExecute:= TRUE );
		iStep := CLIENT_STATE_CLOSE_WAIT;

	CLIENT_STATE_CLOSE_WAIT:
		fbClose( bExecute := FALSE );
		IF NOT fbClose.bBusy THEN

			Connected := FALSE;
			MEMSET( ADR(hSocket), 0, SIZEOF(hSocket));
			IF fbClose.bError THEN

				nErrId := fbClose.nErrId;
				iStep := CLIENT_STATE_ERROR;
			ELSE
				bBusy := FALSE;
				bError := FALSE;
				nErrId := 0;
				iStep := CLIENT_STATE_IDLE;
			END_IF
		END_IF

	CLIENT_STATE_ERROR:
		bError := TRUE;
		IF Connected THEN
			iStep := CLIENT_STATE_CLOSE_START;
		ELSE
			bBusy := FALSE;
			(* iStep := CLIENT_STATE_IDLE *);
		END_IF

END_CASE

END_FUNCTION_BLOCK

// ---- POUs/003_FB/0007_Vacuum/FB_SmcVacuum.TcPOU
FUNCTION_BLOCK FB_SmcVacuum
(*
********************************************************************************
* Name: FB_Encoder
*
* Author:  AutomanH
* Version: 1.0.0
*
* Description:
*   
* Remarks:
*
* Revisions:
* V1.0.0-Automanh Build
* 
*********************************************************************************)
VAR_INPUT
 xIAutoMode:BOOL;
 xIManualMode:BOOL;
 xIVacuumWork:BOOL;//供给阀工作
 xIVacuumBroken:BOOL;//破坏阀工作
 xIVacuumWorkHMI:BOOL;
 xIVacuumBrokenHMI:BOOL;
 xIDeviceRunning:BOOL;
 xIVacuumWorkReached:BOOL;//真空度达到
 xIVacuumBrokenReached:BOOL;//真空以破坏
END_VAR
VAR_OUTPUT
 xQVacuumFeedValve:BOOL;//供给阀输出
 xQVacuumBrokenValve:BOOL;//破坏阀输出
END_VAR

VAR
 VacuumR_TRIG	:	R_TRIG;
VacuumBrokenR_TRIG:R_TRIG;
END_VAR

VacuumR_TRIG(CLK:= ((xIAutoMode OR xIDeviceRunning)AND xIVacuumWork) OR (xIManualMode	AND xIVacuumWorkHMI) , Q=> );
VacuumBrokenR_TRIG(CLK:= ((xIAutoMode OR xIDeviceRunning )AND  xIVacuumBroken) OR (fbMachine[1].xManualMode AND xIVacuumBrokenHMI) , Q=> );
//真空吸
IF	VacuumR_TRIG.Q THEN 
	xQVacuumFeedValve	:= TRUE ;//	卡片搬运工位¶真空发生器1¶供给阀控制
	xQVacuumBrokenValve:=FALSE;//	卡片搬运工位¶真空发生器1¶破坏阀控制
//	xIVacuumWork:=FALSE;
//	xIVacuumWorkHMI:=FALSE;
END_IF 

//真空吸
IF VacuumBrokenR_TRIG.Q THEN 
	xQVacuumBrokenValve	:= TRUE ;
	xQVacuumFeedValve:=FALSE;
//	xIVacuumBroken:=FALSE;
//	xIVacuumBrokenHMI:=FALSE;
END_IF 
IF			xQVacuumBrokenValve AND  xIVacuumBrokenReached THEN
 				xQVacuumBrokenValve	:= FALSE ;
END_IF

	xIVacuumWork:=FALSE;
	xIVacuumWorkHMI:=FALSE;
	xIVacuumBroken:=FALSE;
	xIVacuumBrokenHMI:=FALSE;

END_FUNCTION_BLOCK

// ---- POUs/003_FB/0010_LoadCell/FB_LoadCell.TcPOU
FUNCTION_BLOCK FB_LoadCell EXTENDS FB_Modbus_Tcp
(*
********************************************************************************
* Name: FB_LoadCell
*
* Author:  Automanh
* Version: 1.0.0
*
* Description:
*  LoadSell of XJC-CF3600-F
*
* Remarks:
*
* Revisions:
*   1.0 -AutomanH Rebuild
*********************************************************************************)
VAR_INPUT
xIStart:BOOL;
xIReset:BOOL;
LocalClient:stModbusPara;
stDeviceOpe	:DUT_DeviceOpe;
xIDeviceRunning:BOOL;
xManualMode:BOOL;
xAutoMode:BOOL;
END_VAR
VAR_OUTPUT
 xQRdyCmd:BOOL;
 xQBusy:BOOL;
 xQError:BOOL;
 xQDone:BOOL;
 xQZeroSingle:BOOL;
 stParOut	: ST_LoadCell_ParOut;//参数输出
END_VAR
VAR
	// modbustcp连接步骤
	iCmdStep,iCmdOldStep: INT;
	wLEN:INT;
	wADDR:INT;
	strFunCode:STRING; 
	
	OperR_TRIG:ARRAY[1..20] OF R_TRIG;
	tTimeout:TON;
	tonDelay:TON;
	eErrorID		: ST_LoadCell_Error;(*错误码*)
	// 操作类型
	iOperType: INT;
	i:INT;
	rTempData:REAL;
END_VAR

MEMCPY(ADR(SUPER^.stModbusPara),ADR(LocalClient),SIZEOF(localClient));
SUPER^.M_Modbus();
ACT_Op();
ACT_Cmd();
ACT_Reset();
ACT_Error();

ACTION ACT_Cmd:

IF  NOT  xQBusy THEN
 		xQRdyCmd:=TRUE;
ELSE
 		xQRdyCmd:=FALSE;	
END_IF
tTimeout(IN:= iCmdStep =iCmdOldStep AND iCmdStep<>0 , PT:= T#5S, Q=> , ET=> );
IF		tTimeout.Q THEN
 	xQError:=TRUE;
	eErrorID:=ST_LoadCell_Error.FLT_CMD_TIMEOUT;
END_IF
	 
CASE iCmdStep OF
		0: //等待启动
			 	IF  xIStart THEN
					xQBusy:=TRUE;
					xQDone:=FALSE;
					xIStart:=FALSE;
					iCmdStep:=iCmdStep +1;
				END_IF
		1://等待选择modbusTcp功能码
			 		iCmdOldStep:=iCmdStep;
					iCmdStep:=iCmdStep +1;
		2://判断
					iCmdOldStep:=iCmdStep;
					IF   strFunCode = '10H' THEN
							 tonDelay(IN:= FALSE);
							xQZeroSingle:=TRUE;
							iCmdStep:=iCmdStep +1;
					ELSIF strFunCode = '04H' THEN
					 		iCmdStep:=iCmdStep +2;
					END_IF
					
		3://等待至少20ms以上
				iCmdOldStep:=iCmdStep;
				 tonDelay(IN:= TRUE, PT:=T#100MS , Q=> , ET=> );
				 IF  tonDelay.Q THEN
								 tonDelay(IN:= FALSE);
								xQZeroSingle:=FALSE;
								iCmdStep:=iCmdStep +1;
				 END_IF
		4://读取当前GROSS值
	  					 wQuantityReadInputRegs:=wLEN;(*读取个数*)
	  					 wMBAddReadInputRegs:=wADDR;(*读取起始地址*)
	  					 xReadInputRegs:= TRUE;	
	  				 IF  fbReadInputRegs.bBusy  THEN
	  								xReadInputRegs:=FALSE;
	  							 iCmdOldStep:=iCmdStep;
	  							 iCmdStep:=iCmdStep +1;
	  				 END_IF	
	  5://接收数据
	  	 	iCmdOldStep:=iCmdStep;
	  	 	IF  NOT 	fbReadInputRegs.bBusy AND  NOT  	fbReadInputRegs.bError THEN
				 				MEMCPY(ADR(rTempData),ADR(arwDataReadRegs[1]),SIZEOF(rTempData));
								stParOut.rGROSSWeight:=rTempData;
	  						iCmdStep:=iCmdStep +1;
	  		ELSIF   	fbReadInputRegs.bError THEN
	  					iCmdStep:=0;		
	  					eErrorID:=ST_LoadCell_Error.FLT_PARA;					
	  		END_IF	
		6:
			 		xQDone:=TRUE;
					xQBusy:=FALSE;	 
					iCmdOldStep:=iCmdStep;		
					iCmdStep :=0;					 
END_CASE;
END_ACTION

ACTION ACT_Error:
IF  eErrorID <> 0 THEN
	xQError:=TRUE;
END_IF
//报错内容输出
CASE eErrorID OF 
 	ST_LoadCell_Error.No_ERROR:
		stParOut.sErrorID:='NO ERROR';
	ST_LoadCell_Error.FLT_CMD_TIMEOUT:
		stParOut.sErrorID:='FLT_CMD_TIMEOUT';
	ST_LoadCell_Error.FLT_PARA:
		stParOut.sErrorID:='FLT_PARA';
	
	
END_CASE
END_ACTION

ACTION ACT_OP:
OperR_TRIG[1](CLK:= (xManualMode AND  stDeviceOpe.xReadGROSSHmi) OR((xAutoMode OR  xIDeviceRunning) AND stDeviceOpe.xReadGROSSAuto) , Q=> );	//获取总值GROSS		
OperR_TRIG[2](CLK:= (xManualMode AND  stDeviceOpe.XSetZEROHmi) OR((xAutoMode OR  xIDeviceRunning) AND stDeviceOpe.XSetZEROAuto) , Q=> );		//请零或去皮		
OperR_TRIG[3](CLK:= (xManualMode AND  stDeviceOpe.xSetZEROSaveHmi) OR((xAutoMode OR  xIDeviceRunning) AND stDeviceOpe.xSetZEROSaveAuto) , Q=> );		//保存零点	
OperR_TRIG[13](CLK:=xIReset , Q=> );	//Cancel	
FOR  i:= 1 TO 20 BY 1 DO
 	IF   OperR_TRIG[i].Q THEN
				iOperType:= i;
				xIStart:=TRUE;
				EXIT;
	END_IF
END_FOR

IF   iOperType =1 THEN
  strFunCode:='04H';
 	wLEN := 2;
	wADDR:=0;
ELSIF   iOperType =2 THEN
 	strFunCode:='10H';
	wLEN := 2;
	wADDR:=0;
//由于modbus TCP中不支持10H功能码，所以外接Q点清零
 //	wLEN := 2;
//	wADDR:=4604;
END_IF
stDeviceOpe.xReadGROSSHmi:=stDeviceOpe.xReadGROSSAuto :=FALSE;	//获取总值GROSS
stDeviceOpe.XSetZEROHmi:=stDeviceOpe.XSetZEROAuto		:=FALSE;//去皮或请零
END_ACTION

ACTION ACT_Reset:
IF ( xIReset = TRUE )THEN
 		iCmdStep:=0;
//  	iStep := 0 ;
//		iLoadStep:=0;
  	xQError := FALSE ;
 //	xBusy  := FALSE;
		xQBusy  := FALSE;
//	xStart  := FALSE;
		eErrorID:=MT_MCK_ERROR.No_ERROR;
	  iCmdOldStep:=0;
		xIReset:=FALSE;
END_IF
END_ACTION

END_FUNCTION_BLOCK

// ---- POUs/003_FB/0012_EasyPump/FB_KF300.TcPOU
FUNCTION_BLOCK FB_KF300 EXTENDS FB_Modbus_Tcp
(*
********************************************************************************
* Name: FB_KF300
*
* Author:  Automanh
* Version: 1.0.0
*
* Description:
*  KF300 Control for ShenChen
*
* Remarks:
*
* Revisions:
*   1.0 -AutomanH Rebuild
*********************************************************************************)
VAR_INPUT
	xIReset:BOOL;
	xIManualMode:BOOL;
	xIAutoMode:BOOL;
	xIEstop:BOOL;
	xIDeviceRunning:BOOL;
	LocalClient:stModbusPara;
	stRunPara	:ST_SetPara;//运行参数	
	stDeviceOpe	: stEasyPumpHmi;//操作按钮
END_VAR
VAR_OUTPUT
 	xQRdyCmd:BOOL;
	xQError:BOOL;
	xQBusy:BOOL;
	xQDone:BOOL;
	strQErrorID:STRING;
	xQCalibrationOK:BOOL;
	rMaxRunTime	:REAL;//最大运行时间,单位s
	rMinRunTime	:REAL;//最小运行时间,单位s
END_VAR
VAR
 	xStart:BOOL;
 {attribute 'tc_no_symbol'}
 iParaStep,iOldParaStep,iRunStep,iOldRunStep:INT;
 {attribute 'tc_no_symbol'}
 iCalibStep,iOldCalibStep:INT;
 {attribute 'tc_no_symbol'}
 stLocalPara:ST_LocalPara;
 {attribute 'tc_no_symbol'}
 stPara,stRun,stCalibInit,stCalibAction,stAdjust:ST_StepStatus; 
 {attribute 'tc_no_symbol'}
 stPump:st_EasyPump;
  {attribute 'tc_no_symbol'}
	tTimeout:ARRAY[1..5] OF TON;
 {attribute 'tc_no_symbol'}
	// 蠕动泵读取的液量
	rCurrVolum: REAL;
	{attribute 'tc_no_symbol'}
	//从蠕动泵读取的参数
	stReadPara:ST_ReadPara;
	{attribute 'tc_no_symbol'}
	// 数据数组
	arwData: ARRAY[1..2] OF WORD;
	{attribute 'tc_no_symbol'}
	eErrorID		: PumpError;(*错误码*)
	{attribute 'tc_no_symbol'}
	// 根据设定计算的转速
	rSetSpeed: REAL;
	{attribute 'tc_no_symbol'}
	// 设定的数据
	arwSetData: ARRAY [1..2] OF WORD;
	{attribute 'tc_no_symbol'}
	// 虚拟的较大时间
	rVirtualTime: REAL;
	{attribute 'tc_no_symbol'}
	OperR_TRIG:ARRAY[1..20] OF R_TRIG;
	{attribute 'tc_no_symbol'}
	// 循环计数
	i: INT;
	{attribute 'tc_no_symbol'}
	// 操作类型
	iOperType: INT;
	{attribute 'tc_no_symbol'}
	iOperCounter:INT;
	{attribute 'tc_no_symbol'}
	artDelay:ARRAY[1..5] OF TON;
	{attribute 'tc_no_symbol'}
	tSetTime:TIME;
	tModuleDelay:TON;
	iCalibNum:INT:=1;//校准灌装次数
END_VAR

MEMCPY(ADR(SUPER^.stModbusPara),ADR(LocalClient),SIZEOF(localClient));
SUPER^.M_Modbus();
ACT_RunPara();
ACT_Operation();
ACT_Running();
ACT_ParaCalc();
ACT_Calibration();
ACT_Reset();
ACT_Error();

ACTION ACT_Calibration:
CASE iCalibStep OF
 			0://等待启动
				 IF	stCalibInit.xStart THEN
							stCalibInit.xStart:=FALSE;
							stCalibInit.xBusy:=TRUE;
							stCalibInit.xDone:=FALSE;	
							iCalibStep:=10;//初始化校准参数
				 ELSIF stCalibAction.xStart THEN
						 	 stCalibAction.xStart :=FALSE;
							 stCalibAction.xBusy :=TRUE;
							 stCalibAction.xDone :=FALSE;
							 iCalibStep:=20;//校准
					ELSIF stAdjust.xStart THEN
					 		 stAdjust.xStart :=FALSE;
							 stAdjust.xBusy :=TRUE;
							 stAdjust.xDone :=FALSE;
							 iCalibStep:=30;//微调
				 END_IF
			10://初始化校准参数
					 iOldCalibStep:=iCalibStep;
					 arwDataWriteRegs[1]:=1;
					 wQuantityWriteRegs:=1;
					 wMBAddWriteRegs:=2007;
					 xWriteRegs:=TRUE;
					 IF  fbWriteRegs.bBusy THEN
							 xWriteRegs:=FALSE;
							 iCalibStep:=iCalibStep+1;
					END_IF
			11://液量设定完成
							 iOldCalibStep:=iCalibStep;
						 IF  NOT 	fbWriteRegs.bBusy AND  NOT  	fbWriteRegs.bError THEN
										iCalibStep:=iCalibStep+1;
							ELSIF   	fbReadRegs.bError THEN
									 iCalibStep:=999;				
									 eErrorID:=PumpError.FLT_SET_PARA;					
							END_IF		
		
			12://初始化校准参数完成
						 stCalibInit.xBusy:=FALSE;
							stCalibInit.xDone:=TRUE;	
						 	iCalibStep:=0;
						 
			
			 20://检查实际液量与设定液量的误差范围
					 IF   (stLocalPara.rFluVolumeSet - stLocalPara.iModuleRealVolume )<stLocalPara.rFluVolumeSet*0.5 THEN
							 //误差不能超过0.3ml
							 iCalibStep:=iCalibStep +1;				
					 ELSE
								 eERRORID := PumpError.FLT_Calib_OverFlow;//误差过大
								 iCalibStep:=999;	
					 END_IF
			 21://需要设定实际液量--实际液量最好是三组液量的平均值
							iOldCalibStep:=iCalibStep;
							MEMCPY(ADR(arwSetData[1]),ADR(stLocalPara.iModuleRealVolume),SIZEOF(stLocalPara.iModuleRealVolume) ); 
							arwDataWriteRegs[1]:=arwSetData[2];
							arwDataWriteRegs[2]:=arwSetData[1];
							wQuantityWriteRegs:=2;
							wMBAddWriteRegs:=2004;
							xWriteRegs:=TRUE;
							IF  fbWriteRegs.bBusy THEN
									xWriteRegs:=FALSE;
									 iCalibStep:=iCalibStep +1;		
						 END_IF
			 22://液量设定完成
							iOldCalibStep:=iCalibStep;
						 IF  NOT 	fbWriteRegs.bBusy AND  NOT  	fbWriteRegs.bError THEN
											 iCalibStep:=iCalibStep +1;		
							ELSIF   	fbReadRegs.bError THEN
										 iCalibStep:=999;				
										 eErrorID:=PumpError.FLT_CALIB_PARA;					
							END_IF		
			 23://校准实际液量设定结束
						 stCalibAction.xBusy :=FALSE;
						 stCalibAction.xDone :=TRUE;
						 iCalibStep:=0;				 
			30://校准微调-微调幅度为(设定量*0.001),这里要根据客户要求的精度进行调整
					 xQCalibrationOK:=FALSE;
					 iCalibStep:=iCalibStep +1;
			31://检测数据是否在精度范围内
					 iOldCalibStep:=iCalibStep;
					 IF  stLocalPara.iModuleRealVolume>=stLocalPara.rFluVolumeSet-(stLocalPara.rFluVolumeSet*stLocalPara.iAccuracySet) AND 
							 stLocalPara.iModuleRealVolume<=stLocalPara.rFluVolumeSet+(stLocalPara.rFluVolumeSet*stLocalPara.iAccuracySet) THEN
							 	 xQCalibrationOK:=TRUE;
								 iCalibStep:=36;
					ELSIF stLocalPara.iModuleRealVolume>=stLocalPara.rFluVolumeSet-(stLocalPara.rFluVolumeSet*stLocalPara.iAccuracySet) THEN
								 iCalibStep:=iCalibStep +1;	//需要减小
					ELSIF  stLocalPara.iModuleRealVolume<=stLocalPara.rFluVolumeSet+(stLocalPara.rFluVolumeSet*stLocalPara.iAccuracySet) THEN
								 iCalibStep:=iCalibStep +3;	//需要增大
					END_IF
			32://发送微调指令
					iOldParaStep:=iParaStep;
					arwDataWriteRegs[1]:=0;
					wQuantityWriteRegs:=1;
					wMBAddWriteRegs:=2006;
					xWriteRegs:=TRUE;
					IF  fbWriteRegs.bBusy THEN
							xWriteRegs:=FALSE;
							iCalibStep:=iCalibStep+1;
				 END_IF
		  33://微调执行完成
					 iOldParaStep:=iParaStep;
					 IF  NOT 	fbWriteRegs.bBusy AND  NOT  	fbWriteRegs.bError THEN
									 iCalibStep:=36;
						ELSIF   	fbReadRegs.bError THEN
								 iCalibStep:=999;				
								 eErrorID:=PumpError.FLT_SET_PARA;					
						END_IF			 
			34://发送微调指令
					iOldParaStep:=iParaStep;
					arwDataWriteRegs[1]:=1;
					wQuantityWriteRegs:=1;
					wMBAddWriteRegs:=2006;
					xWriteRegs:=TRUE;
					IF  fbWriteRegs.bBusy THEN
							xWriteRegs:=FALSE;
							iCalibStep:=iCalibStep+1;
				 END_IF
		  35://微调执行完成
					 iOldParaStep:=iParaStep;
					 IF  NOT 	fbWriteRegs.bBusy AND  NOT  	fbWriteRegs.bError THEN
									 iCalibStep:=36;
						ELSIF   	fbReadRegs.bError THEN
								 iCalibStep:=999;				
								 eErrorID:=PumpError.FLT_SET_PARA;					
						END_IF			 			
			 36://微调完成
							 stAdjust.xBusy :=FALSE;
							 stAdjust.xDone :=TRUE;
							 iCalibStep:=0;//校准			
END_CASE
 //防止程序二次执行
 IF	stCalibInit.xBusy THEN
			stCalibInit.xStart:=FALSE;
 ELSIF stCalibAction.xBusy THEN
			stCalibAction.xStart :=FALSE;
 ELSIF stAdjust.xBusy THEN
			stAdjust.xStart :=FALSE;
 END_IF
END_ACTION

ACTION ACT_Error:
tTimeout[1](IN:= iParaStep =iOldParaStep AND iParaStep<>0 , PT:= T#15S, Q=> , ET=> );
tTimeout[2](IN:= iRunStep =iOldRunStep AND iRunStep<>0 , PT:= T#15S, Q=> , ET=> );
tTimeout[3](IN:= iCalibStep =iOldCalibStep AND iCalibStep<>0 , PT:= T#15S, Q=> , ET=> );
IF		tTimeout[1].Q THEN
	  	stPara.xError:=TRUE;
	  	stPara.xBusy:=FALSE;
			eErrorID:=PumpError.FLT_CMD_TIMEOUT;
	    iParaStep := 999;
END_IF

IF		tTimeout[2].Q THEN
			stRun.xError:=TRUE;
			stRun.xBusy:=FALSE;
			eErrorID:=PumpError.FLT_CMD_TIMEOUT;
			iRunStep := 999;
END_IF

IF		tTimeout[3].Q THEN
			stAdjust.xError:=TRUE;
			stAdjust.xBusy:=FALSE;
			eErrorID:=PumpError.FLT_CMD_TIMEOUT;
			iCalibStep := 999;
END_IF

IF  eErrorID <> PumpError.NO_ERROR THEN
		xQError:=TRUE;
END_IF
//报错内容输出
CASE eErrorID OF 
		 PumpError.No_ERROR:
			 strQErrorID:='NO ERROR';
		 PumpError.FLT_PARA:
			 strQErrorID:='FLT_PARA';
		 PumpError.FLT_FLUVOLUM_TIME_PARA:
			 strQErrorID:='FLT_FLUVOLUM_TIME_PARA';
		 PumpError.FLT_SET_PARA:
			 strQErrorID:='FLT_SET_PARA';	
		 PumpError.FLT_CMD_TIMEOUT:
			 strQErrorID:='FLT_CMD_TIMEOUT';	
		 PumpError.FLT_RUN_ERROR:
			 strQErrorID:='FLT_RUN_ERROR';
		 PumpError.FLT_Calib_OverFlow:
			 strQErrorID:='FLT_Calib_OverFlow';	
		 PumpError.FLT_CALIB_PARA:
			 strQErrorID:='FLT_CALIB_PARA';		
		 PumpError.FLT_CONFIGURE_PARA:
			 strQErrorID:='FLT_CONFIGURE_PARA';		
END_CASE
END_ACTION

ACTION ACT_Operation:
OperR_TRIG[1](CLK:= (xIManualMode AND  stDeviceOpe.xPush_Hmi[1]) OR((xIAutoMode OR  xIDeviceRunning) AND stDeviceOpe.xPush_Auto[1]) , Q=> );	//Push
OperR_TRIG[2](CLK:= (xIManualMode AND  stDeviceOpe.xPush_Hmi[2]) OR((xIAutoMode OR  xIDeviceRunning) AND stDeviceOpe.xPush_Auto[2]) , Q=> );	//Push
OperR_TRIG[3](CLK:= (xIManualMode AND  stDeviceOpe.xPush_Hmi[3]) OR((xIAutoMode OR  xIDeviceRunning) AND stDeviceOpe.xPush_Auto[3]) , Q=> );	//Push
OperR_TRIG[4](CLK:= (xIManualMode AND  stDeviceOpe.xPush_Hmi[4]) OR((xIAutoMode OR  xIDeviceRunning) AND stDeviceOpe.xPush_Auto[4]) , Q=> );	//Push
OperR_TRIG[5](CLK:= (xIManualMode AND  stDeviceOpe.xPush_Hmi[5]) OR((xIAutoMode OR  xIDeviceRunning) AND stDeviceOpe.xPush_Auto[5]) , Q=> );	//Push
OperR_TRIG[6](CLK:= (xIManualMode AND  stDeviceOpe.xPull_Hmi[1]) OR((xIAutoMode OR  xIDeviceRunning) AND stDeviceOpe.xPull_Auto[1]) , Q=> );	//Pull
OperR_TRIG[7](CLK:= (xIManualMode AND  stDeviceOpe.xPull_Hmi[2]) OR((xIAutoMode OR  xIDeviceRunning) AND stDeviceOpe.xPull_Auto[2]) , Q=> );	//Pull
OperR_TRIG[8](CLK:= (xIManualMode AND  stDeviceOpe.xPull_Hmi[3]) OR((xIAutoMode OR  xIDeviceRunning) AND stDeviceOpe.xPull_Auto[3]) , Q=> );	//Pull
OperR_TRIG[9](CLK:= (xIManualMode AND  stDeviceOpe.xPull_Hmi[4]) OR((xIAutoMode OR  xIDeviceRunning) AND stDeviceOpe.xPull_Auto[4]) , Q=> );	//Pull
OperR_TRIG[10](CLK:= (xIManualMode AND  stDeviceOpe.xPull_Hmi[5]) OR((xIAutoMode OR  xIDeviceRunning) AND stDeviceOpe.xPull_Auto[5]) , Q=> );	//Pull
OperR_TRIG[11](CLK:= (xIManualMode AND  stDeviceOpe.xModulePush_Hmi) OR((xIAutoMode OR  xIDeviceRunning) AND stDeviceOpe.xModulePush_Auto) , Q=> );		//ModulePush	
OperR_TRIG[12](CLK:= (xIManualMode AND  stDeviceOpe.xFullSpeedPush_Hmi) OR((xIAutoMode OR  xIDeviceRunning) AND stDeviceOpe.xFullSpeedPush_Auto) , Q=> );//FullSpeedPush
OperR_TRIG[13](CLK:= (xIManualMode AND  stDeviceOpe.xFullSpeedPull_Hmi) OR((xIAutoMode OR  xIDeviceRunning) AND stDeviceOpe.xFullSpeedPull_Auto) , Q=> );//FullSpeedPull
OperR_TRIG[14](CLK:= (xIManualMode AND  stDeviceOpe.xFullSpeedStop_Hmi) OR((xIAutoMode OR  xIDeviceRunning) AND stDeviceOpe.xFullSpeedStop_Auto) , Q=> );//FullSpeedStop
OperR_TRIG[15](CLK:= (xIManualMode AND  stDeviceOpe.xStop_Hmi) OR((xIAutoMode OR  xIDeviceRunning) AND stDeviceOpe.xStop_Auto  ) , Q=> );//Stop
OperR_TRIG[16](CLK:= (xIManualMode AND  stDeviceOpe.xCalibAction_Hmi) OR((xIAutoMode OR  xIDeviceRunning) AND stDeviceOpe.xCalibAction_Auto) , Q=> );//Calibration Action
OperR_TRIG[17](CLK:= (xIManualMode AND  stDeviceOpe.xCalibInit_Hmi) OR((xIAutoMode OR  xIDeviceRunning) AND stDeviceOpe.xCalibInit_Auto), Q=> );//Calibration Init
OperR_TRIG[18](CLK:= (xIManualMode AND  stDeviceOpe.xAdjust_Hmi) OR((xIAutoMode OR  xIDeviceRunning) AND stDeviceOpe.xAdjust_Auto), Q=> );//Adjust
OperR_TRIG[19](CLK:= xIEstop, Q=> );//Estop

FOR  i:= 1 TO 20 BY 1 DO
 	IF   OperR_TRIG[i].Q THEN
				iOperCounter:= i;
				xStart:=TRUE;
				EXIT;
	END_IF
END_FOR
//Push
FOR  i:=1 TO 5 BY 1 DO
 		IF   iOperCounter =i THEN
		 		stLocalPara.rFluVolumeSet	:=stRunPara.rPushFluVolume[i];
				stLocalPara.rRuntimeSet	:=stRunPara.rPushRuntime[i];
				stLocalPara.iCycleNumber	:=stRunPara.iPushCycleNumber[i];
				stLocalPara.iBackAngle:=stRunPara.iPushBackAngle[i];
				stLocalPara.iDirectionSet:=stRunPara.iDirectionSet;
				stLocalPara.rVirualTime:=rMaxRunTime -1;
				iOperType:=stOperType.iPush;
		END_IF
END_FOR
//pull
FOR  i:=6 TO 10 BY 1 DO
 		IF   iOperCounter =i THEN
		 		stLocalPara.rFluVolumeSet	:=stRunPara.rPullFluVolume[i-5];
				stLocalPara.rRuntimeSet	:=stRunPara.rPullRuntime[i-5];
				stLocalPara.iCycleNumber	:=stRunPara.iPullCycleNumber[i-5];
				stLocalPara.iBackAngle:=stRunPara.iPullBackAngle[i-5];
				stLocalPara.iDirectionSet:=ABS(1-stRunPara.iDirectionSet);
				stLocalPara.rVirualTime:=rMaxRunTime -1;
				iOperType:=stOperType.iPull;
		END_IF
END_FOR 
 //Module Push
IF   iOperCounter =11 THEN
		 		stLocalPara.rFluVolumeSet	:=stRunPara.rCalFluVolume;
				stLocalPara.rRuntimeSet	 :=stRunPara.rCalTime;
				stLocalPara.iCycleNumber :=stRunPara.rCalNum;
				stLocalPara.iBackAngle:=stRunPara.rCalBackAngle;
				stLocalPara.iDirectionSet:=stRunPara.iDirectionSet;
				stLocalPara.iModuleAdress:=stRunPara.iModuleAdress;
				stLocalPara.iModuleSpeed:= stRunPara.rCalFluVolume * 60.0/(stRunPara.rSpeedRatio* stRunPara.rCalTime);
				stLocalPara.rVirualTime:=rMaxRunTime -1;
				iOperType:=stOperType.iModulePush;
////FullSpeedPush
ELSIF  iOperCounter =12 THEN
 				stLocalPara.iDirectionSet:=stRunPara.iDirectionSet;
 				iOperType:=stOperType.iFullSpeedPush;
ELSIF  iOperCounter =13 THEN
 			stLocalPara.iDirectionSet:=ABS(1-stRunPara.iDirectionSet);
 			iOperType:=stOperType.iFullSpeedPull;
ELSIF  iOperCounter =14 THEN
 			iOperType:=stOperType.iFullSpeedStop;
ELSIF  iOperCounter =15 OR iOperCounter =19  THEN
 			iOperType:=stOperType.iStop;
ELSIF  iOperCounter =16  THEN//Calibration
 			stLocalPara.iModuleRealVolume:=stRunPara.rModuleRealFluVolume;
 			iOperType:=stOperType.iCalibAction;
ELSIF  iOperCounter =17  THEN
 			iOperType:=stOperType.iCalibInit;	
ELSIF    iOperCounter =18 THEN //adjust
 			stLocalPara.iModuleRealVolume:=stRunPara.rModuleRealFluVolume;
 			stLocalPara.iAccuracySet:=stRunPara.iAccuracySet;
 			iOperType:=stOperType.iAdjust;	
END_IF


MEMSET(ADR(stDeviceOpe),0,SIZEOF(stDeviceOpe));
END_ACTION

ACTION ACT_ParaCalc:
//
(*************************检测配置参数是否匹配成功*********************************)
IF stRunPara.iPumpType=RudongPump_PumpType.DFPluse THEN
	//MiniPump泵头
	IF  stRunPara.iPumpTypeSet=RudongPump_PumpHeadType.MiniPump01 THEN
		stPump.iPumpType:=0;//泵头值为0
			IF stRunPara.iHosePipeTypeSet=RudongPump_SoftPipeType.P13 THEN//13#软管
				stPump.iHosePipeType:=13;//软管类型值13
				IF  stLocalPara.rFluVolumeSet*1000/135<0.1 THEN
					rMaxRunTime:=	0.1;
				ELSE
					rMaxRunTime:=	stLocalPara.rFluVolumeSet*1000/135;
				END_IF
				rMaxRunTime:=	(stLocalPara.rFluVolumeSet/0.45)*0.2;//最大流量(0.45微升/秒,0.0024ml/min)	
			ELSIF stRunPara.iHosePipeTypeSet=RudongPump_SoftPipeType.P14 THEN//14#软管
					stPump.iHosePipeType:=13;//软管类型值13
				IF stLocalPara.rFluVolumeSet*1000/570<0.1 THEN
							rMinRunTime:=	0.1;
				ELSE
						rMinRunTime:=	stLocalPara.rFluVolumeSet*1000/135;
				END_IF
				rMaxRunTime:=	(stLocalPara.rFluVolumeSet/1.9)*0.2;	
			ELSIF stRunPara.iHosePipeTypeSet=RudongPump_SoftPipeType.P19 THEN//19#软管
				stPump.iHosePipeType:=19;
				IF stLocalPara.rFluVolumeSet*1000/1240<0.1 THEN
					rMinRunTime:=	0.1;
				ELSE
					rMinRunTime:=	stLocalPara.rFluVolumeSet*1000/1240;
				END_IF
					rMaxRunTime:=	(stLocalPara.rFluVolumeSet*1000/4.13)*0.2;		
			ELSIF stRunPara.iHosePipeTypeSet=RudongPump_SoftPipeType.P16 THEN//16#软管
					stPump.iHosePipeType:=16;
				IF stLocalPara.rFluVolumeSet*1000/1880<0.1 THEN
					rMinRunTime:=	0.1;
				ELSE
					rMinRunTime:=	stLocalPara.rFluVolumeSet*1000/1880;
				END_IF
				rMaxRunTime:=	(stLocalPara.rFluVolumeSet*1000/6.28)*0.2;	
			ELSIF stRunPara.iHosePipeTypeSet=RudongPump_SoftPipeType.P25 THEN//25#软管
					stPump.iHosePipeType:=25;
				IF stLocalPara.rFluVolumeSet*1000/3100<0.1 THEN
					rMinRunTime:=	0.1;
				ELSE
					rMinRunTime:=	stLocalPara.rFluVolumeSet*1000/3100;
				END_IF
				rMaxRunTime:=	(stLocalPara.rFluVolumeSet*1000/10.33)*0.2;			
		ELSE
				eERRORID:=RudongPump_ERROR.FLT_CONFIGURE_PARA;		
		END_IF
	//UD15
	ELSIF  stRunPara.iPumpTypeSet=RudongPump_PumpHeadType.UD15 THEN
				stPump.iHosePipeType:=1;//泵头值为0
			IF stRunPara.iHosePipeTypeSet=RudongPump_SoftPipeType.P16 THEN//16#软管
				stPump.iHosePipeType:=16;
				IF stLocalPara.rFluVolumeSet*1000/4000<0.1 THEN
					rMinRunTime:=	0.1;
				ELSE
					rMinRunTime:=	stLocalPara.rFluVolumeSet*1000/4000;
				END_IF
				rMaxRunTime:=	(stLocalPara.rFluVolumeSet*1000/13.33)*0.2;		
			ELSIF stRunPara.iHosePipeTypeSet=RudongPump_SoftPipeType.P17 THEN//17#软管
				stPump.iHosePipeType:=17;
				IF stLocalPara.rFluVolumeSet*1000/15000<0.1 THEN
					rMinRunTime:=	0.1;
				ELSE
					rMinRunTime:=	stLocalPara.rFluVolumeSet*1000/15000;
				END_IF
				rMaxRunTime:=	(stLocalPara.rFluVolumeSet*1000/50)*0.2;	
			ELSIF stRunPara.iHosePipeTypeSet=RudongPump_SoftPipeType.P25 THEN//25#软管
				stPump.iHosePipeType:=25;
				IF stLocalPara.rFluVolumeSet*1000/8000<0.1 THEN
					rMinRunTime:=	0.1;
				ELSE
					rMinRunTime:=	stLocalPara.rFluVolumeSet*1000/8000;
				END_IF
				 rMaxRunTime:=	(stLocalPara.rFluVolumeSet*1000/26.66)*0.2;			
		ELSE
				eERRORID:=RudongPump_ERROR.FLT_CONFIGURE_PARA;		
		END_IF
	//HandyPump01泵头
ELSIF  stRunPara.iPumpTypeSet=RudongPump_PumpHeadType.HandyPump01 THEN
 			IF stRunPara.iHosePipeTypeSet=RudongPump_SoftPipeType.P13 THEN//13#软管,三滚轮
				IF stLocalPara.rFluVolumeSet*1000/155<0.1 THEN
					rMinRunTime:=	0.1;
				ELSE
					rMinRunTime:=	stLocalPara.rFluVolumeSet*1000/155;
				END_IF
					rMaxRunTime:=	(stLocalPara.rFluVolumeSet*1000/0.51)*0.2;	
		
	(*	IF stRunPara.iHosePipeTypeSet=RudongPump_SoftPipeType.P13 THEN//13#软管,三滚轮
			iMinRunTime:=	(rFluVolumeSet/10)*60;
			iMaxRunTime:=	(rFluVolumeSet/0.0033)*60;	
		ELSIF stRunPara.iHosePipeTypeSet=RudongPump_SoftPipeType.P14 THEN//14#软管,三滚轮
			iMinRunTime:=	(rFluVolumeSet/56)*60;
			iMaxRunTime:=	(rFluVolumeSet/0.0187)*60;		
		ELSIF stRunPara.iHosePipeTypeSet=RudongPump_SoftPipeType.P19 THEN//19#软管,三滚轮
			iMinRunTime:=	(rFluVolumeSet/111)*60;
			iMaxRunTime:=	(rFluVolumeSet/0.0371)*60;
		ELSIF stRunPara.iHosePipeTypeSet=RudongPump_SoftPipeType.P16 THEN//16#软管,三滚轮
			iMinRunTime:=	(rFluVolumeSet/190)*60;
			iMaxRunTime:=	(rFluVolumeSet/0.0636)*60;		
		ELSIF stRunPara.iHosePipeTypeSet=RudongPump_SoftPipeType.P25 THEN//25#软管,三滚轮
			iMinRunTime:=	(rFluVolumeSet/365)*60;
			iMaxRunTime:=	(rFluVolumeSet/0.1219)*60;
	*)
		ELSE
				eERRORID:=RudongPump_ERROR.FLT_CONFIGURE_PARA;						
		END_IF
	END_IF
ELSE
		eERRORID:=RudongPump_ERROR.FLT_CONFIGURE_PARA;
END_IF


(*
//MiniPump01泵头
IF  stRunPara.iPumpTypeSet=RudongPump_PumpHeadType.MiniPump01 THEN
		IF stRunPara.iHosePipeTypeSet=RudongPump_SoftPipeType.P13 THEN//13#软管
			iMinRunTime:=	(rFluVolumeSet/8)*60;//最大流量(135微升/秒,8.28ml/min)
			iMaxRunTime:=	(rFluVolumeSet/0.45)*60;//最大流量(0.45微升/秒,0.0024ml/min)	
		ELSIF stRunPara.iHosePipeTypeSet=RudongPump_SoftPipeType.P14 THEN//14#软管
			iMinRunTime:=	(rFluVolumeSet/33)*60;
			iMaxRunTime:=	(rFluVolumeSet/1.9)*60;
		ELSIF stRunPara.iHosePipeTypeSet=RudongPump_SoftPipeType.P19 THEN//19#软管
			iMinRunTime:=	(rFluVolumeSet/77)*60;
			iMaxRunTime:=	(rFluVolumeSet/4.13)*60;	
		ELSIF stRunPara.iHosePipeTypeSet=RudongPump_SoftPipeType.P16 THEN//16#软管
			iMinRunTime:=	(rFluVolumeSet/114)*60;
			iMaxRunTime:=	(rFluVolumeSet/6.28)*60;	
		ELSIF stRunPara.iHosePipeTypeSet=RudongPump_SoftPipeType.P25 THEN//25#软管
			iMinRunTime:=	(rFluVolumeSet/190)*60;
			iMaxRunTime:=	(rFluVolumeSet/10.33)*60;		
		ELSIF stRunPara.iHosePipeTypeSet=RudongPump_SoftPipeType.P1_1 THEN//1x1#软管
			iMinRunTime:=	(rFluVolumeSet/15)*60;
			iMaxRunTime:=	(rFluVolumeSet/4.5)*60;	
		ELSIF stRunPara.iHosePipeTypeSet=RudongPump_SoftPipeType.P2_1 THEN//2x1#软管
			iMinRunTime:=	(rFluVolumeSet/54)*60;
			iMaxRunTime:=	(rFluVolumeSet/4.5)*60;		
		ELSIF stRunPara.iHosePipeTypeSet=RudongPump_SoftPipeType.P2_5_1 THEN//2.5x1#软管
			iMinRunTime:=	(rFluVolumeSet/76)*60;
			iMaxRunTime:=	(rFluVolumeSet/5)*60;		
		ELSIF stRunPara.iHosePipeTypeSet=RudongPump_SoftPipeType.P3_1 THEN//3x1#软管
			iMinRunTime:=	(rFluVolumeSet/108)*60;
			iMaxRunTime:=	(rFluVolumeSet/5)*60;
	ELSE
			eERRORID:=RudongPump_ERROR.FLT_CONFIGURE_PARA;		
	END_IF		
	
//MiniPump02泵头
ELSIF  stRunPara.iPumpTypeSet=RudongPump_PumpHeadType.MiniPump02 THEN
	IF stRunPara.iHosePipeTypeSet=RudongPump_SoftPipeType.P1_1 THEN//1x1#软管
		iMinRunTime:=	(rFluVolumeSet/15.01)*60;
		iMaxRunTime:=	(rFluVolumeSet/0.005)*60;	
	ELSIF stRunPara.iHosePipeTypeSet=RudongPump_SoftPipeType.P2_1 THEN//2x1#软管
		iMinRunTime:=	(rFluVolumeSet/54.63)*60;
		iMaxRunTime:=	(rFluVolumeSet/0.018)*60;		
	ELSIF stRunPara.iHosePipeTypeSet=RudongPump_SoftPipeType.P2_5_1 THEN//2.5x1#软管
		iMinRunTime:=	(rFluVolumeSet/76.84)*60;
		iMaxRunTime:=	(rFluVolumeSet/0.0256)*60;
	ELSE
			eERRORID:=RudongPump_ERROR.FLT_CONFIGURE_PARA;						
	END_IF	

//HandyPump01泵头
ELSIF  stRunPara.iPumpTypeSet=RudongPump_PumpHeadType.HandyPump01 THEN
	IF stRunPara.iHosePipeTypeSet=RudongPump_SoftPipeType.P13 THEN//13#软管,三滚轮
		iMinRunTime:=	(rFluVolumeSet/10)*60;
		iMaxRunTime:=	(rFluVolumeSet/0.0033)*60;	
	ELSIF stRunPara.iHosePipeTypeSet=RudongPump_SoftPipeType.P14 THEN//14#软管,三滚轮
		iMinRunTime:=	(rFluVolumeSet/56)*60;
		iMaxRunTime:=	(rFluVolumeSet/0.0187)*60;		
	ELSIF stRunPara.iHosePipeTypeSet=RudongPump_SoftPipeType.P19 THEN//19#软管,三滚轮
		iMinRunTime:=	(rFluVolumeSet/111)*60;
		iMaxRunTime:=	(rFluVolumeSet/0.0371)*60;
	ELSIF stRunPara.iHosePipeTypeSet=RudongPump_SoftPipeType.P16 THEN//16#软管,三滚轮
		iMinRunTime:=	(rFluVolumeSet/190)*60;
		iMaxRunTime:=	(rFluVolumeSet/0.0636)*60;		
	ELSIF stRunPara.iHosePipeTypeSet=RudongPump_SoftPipeType.P25 THEN//25#软管,三滚轮
		iMinRunTime:=	(rFluVolumeSet/365)*60;
		iMaxRunTime:=	(rFluVolumeSet/0.1219)*60;
	ELSE
			eERRORID:=RudongPump_ERROR.FLT_CONFIGURE_PARA;						
	END_IF

//HandyPump02泵头
ELSIF  stRunPara.iPumpTypeSet=RudongPump_PumpHeadType.HandyPump02 THEN
	IF stRunPara.iHosePipeTypeSet=RudongPump_SoftPipeType.P13 THEN//13#软管,三滚轮
		iMinRunTime:=	(rFluVolumeSet/10)*60;
		iMaxRunTime:=	(rFluVolumeSet/0.0033)*60;	
	ELSIF stRunPara.iHosePipeTypeSet=RudongPump_SoftPipeType.P14 THEN//14#软管,三滚轮
		iMinRunTime:=	(rFluVolumeSet/56)*60;
		iMaxRunTime:=	(rFluVolumeSet/0.0187)*60;		
	ELSIF stRunPara.iHosePipeTypeSet=RudongPump_SoftPipeType.P19 THEN//19#软管,三滚轮
		iMinRunTime:=	(rFluVolumeSet/111)*60;
		iMaxRunTime:=	(rFluVolumeSet/0.0371)*60;
	ELSIF stRunPara.iHosePipeTypeSet=RudongPump_SoftPipeType.P16 THEN//16#软管,三滚轮
		iMinRunTime:=	(rFluVolumeSet/190)*60;
		iMaxRunTime:=	(rFluVolumeSet/0.0636)*60;	
	ELSE
			eERRORID:=RudongPump_ERROR.FLT_CONFIGURE_PARA;							
	END_IF

//EasyPumpI_III泵头,单通道
ELSIF  stRunPara.iPumpTypeSet=RudongPump_PumpHeadType.EasyPumpI_III THEN
	IF stRunPara.iHosePipeTypeSet=RudongPump_SoftPipeType.P13 THEN//13#软管
		iMinRunTime:=	(rFluVolumeSet/32)*60;
		iMaxRunTime:=	(rFluVolumeSet/0.0053)*60;	
	ELSIF stRunPara.iHosePipeTypeSet=RudongPump_SoftPipeType.P14 THEN//14#软管
		iMinRunTime:=	(rFluVolumeSet/162)*60;
		iMaxRunTime:=	(rFluVolumeSet/0.027)*60;		
	ELSIF stRunPara.iHosePipeTypeSet=RudongPump_SoftPipeType.P19 THEN//19#软管
		iMinRunTime:=	(rFluVolumeSet/330)*60;
		iMaxRunTime:=	(rFluVolumeSet/0.055)*60;
	ELSIF stRunPara.iHosePipeTypeSet=RudongPump_SoftPipeType.P16 THEN//16#软管
		iMinRunTime:=	(rFluVolumeSet/560)*60;
		iMaxRunTime:=	(rFluVolumeSet/0.093)*60;	
	ELSIF stRunPara.iHosePipeTypeSet=RudongPump_SoftPipeType.P25 THEN//25#软管
		iMinRunTime:=	(rFluVolumeSet/1180)*60;
		iMaxRunTime:=	(rFluVolumeSet/0.197)*60;	
	ELSIF stRunPara.iHosePipeTypeSet=RudongPump_SoftPipeType.P17 THEN//17#软管
		iMinRunTime:=	(rFluVolumeSet/2000)*60;
		iMaxRunTime:=	(rFluVolumeSet/0.333)*60;	
	ELSIF stRunPara.iHosePipeTypeSet=RudongPump_SoftPipeType.P18 THEN//18#软管
		iMinRunTime:=	(rFluVolumeSet/2580)*60;
		iMaxRunTime:=	(rFluVolumeSet/0.430)*60;	
	ELSE
			eERRORID:=RudongPump_ERROR.FLT_CONFIGURE_PARA;							
	END_IF

//EasyPumpII_IV泵头,单通道
ELSIF  stRunPara.iPumpTypeSet=RudongPump_PumpHeadType.EasyPumpII_IV THEN
	IF stRunPara.iHosePipeTypeSet=RudongPump_SoftPipeType.P15 THEN//15#软管
		iMinRunTime:=	(rFluVolumeSet/1080)*60;
		iMaxRunTime:=	(rFluVolumeSet/0.0180)*60;	
	ELSIF stRunPara.iHosePipeTypeSet=RudongPump_SoftPipeType.P24 THEN//24#软管
		iMinRunTime:=	(rFluVolumeSet/1640)*60;
		iMaxRunTime:=	(rFluVolumeSet/0.273)*60;		
	ELSIF stRunPara.iHosePipeTypeSet=RudongPump_SoftPipeType.P35 THEN//35#软管
		iMinRunTime:=	(rFluVolumeSet/2300)*60;
		iMaxRunTime:=	(rFluVolumeSet/0.383)*60;
	ELSIF stRunPara.iHosePipeTypeSet=RudongPump_SoftPipeType.P36 THEN//36#软管
		iMinRunTime:=	(rFluVolumeSet/3100)*60;
		iMaxRunTime:=	(rFluVolumeSet/0.517)*60;	
	ELSE
			eERRORID:=RudongPump_ERROR.FLT_CONFIGURE_PARA;							
	END_IF

//EasyPumpV_VI泵头,双通道
ELSIF  stRunPara.iPumpTypeSet=RudongPump_PumpHeadType.EasyPumpV_VI THEN
		IF stRunPara.iHosePipeTypeSet=RudongPump_SoftPipeType.P13 THEN//13#软管
		iMinRunTime:=	(rFluVolumeSet/32)*60;
		iMaxRunTime:=	(rFluVolumeSet/0.0053)*60;	
	ELSIF stRunPara.iHosePipeTypeSet=RudongPump_SoftPipeType.P14 THEN//14#软管
		iMinRunTime:=	(rFluVolumeSet/162)*60;
		iMaxRunTime:=	(rFluVolumeSet/0.0027)*60;		
	ELSIF stRunPara.iHosePipeTypeSet=RudongPump_SoftPipeType.P19 THEN//19#软管
		iMinRunTime:=	(rFluVolumeSet/330)*60;
		iMaxRunTime:=	(rFluVolumeSet/0.0055)*60;
	ELSIF stRunPara.iHosePipeTypeSet=RudongPump_SoftPipeType.P16 THEN//16#软管
		iMinRunTime:=	(rFluVolumeSet/560)*60;
		iMaxRunTime:=	(rFluVolumeSet/0.093)*60;		
	ELSIF stRunPara.iHosePipeTypeSet=RudongPump_SoftPipeType.P25 THEN//25#软管
		iMinRunTime:=	(rFluVolumeSet/1180)*60;
		iMaxRunTime:=	(rFluVolumeSet/0.197)*60;
	ELSE
			eERRORID:=RudongPump_ERROR.FLT_CONFIGURE_PARA;							
	END_IF
	
END_IF


END_IF

*)
		


//参数超出范围报错	
IF stLocalPara.rFluVolumeSet<>0 THEN
	IF stLocalPara.rRuntimeSet<rMinRunTime OR stLocalPara.rRuntimeSet>rMaxRunTime OR  rMaxRunTime<rMinRunTime THEN
		eERRORID:=RudongPump_ERROR.FLT_CONFIGURE_PARA;
	END_IF
END_IF
END_ACTION

ACTION ACT_Reset:
IF   xIReset THEN
 
 	 iParaStep:=0;
	 iRunStep:=0;
 	 iCalibStep:=0;
	 
	 iOldParaStep:=0;
	 iOldRunStep:=0;
	 iOldCalibStep:=0;
	 
	 stPara.xStart:=FALSE;
	 stPara.xBusy:=FALSE;
	 stPara.xError:=FALSE;
 
	 stRun.xStart:=FALSE;
	 stRun.xBusy:=FALSE;
	 stRun.xError:=FALSE;
		
	 stCalibInit.xStart:=FALSE;
	 stCalibInit.xBusy:=FALSE;
	 stCalibInit.xDone:=FALSE;
	 
	 stCalibAction.xStart:=FALSE;
	 stCalibAction.xBusy :=FALSE;
	 stCalibAction.xDone :=FALSE;
	 
	 stAdjust.xStart:=FALSE;
	 stAdjust.xBusy :=FALSE;
	 stAdjust.xDone :=FALSE;
	 
	
	 
	 xQBusy:=FALSE;
	 //xQDone:=FALSE;
	 
	 eErrorID := PumpError.NO_ERROR;
	 xIReset:=FALSE;
END_IF
END_ACTION

ACTION ACT_Running:
IF  NOT  xQBusy THEN
 		xQRdyCmd:=TRUE;
ELSE
 		xQRdyCmd:=FALSE;	
END_IF

CASE  iRunStep OF 
 0://等待开始
 		IF  xStart THEN
		 		xStart:=FALSE;
				xQBusy:=TRUE;
				xQDone:=FALSE;
				iRunStep:=iRunStep +1;
		END_IF
 1://检查是否是全速
 		IF    iOperType=stOperType.iFullSpeedPull OR 
					iOperType=stOperType.iFullSpeedPush OR
					iOperType=stOperType.iStop OR
					iOperType=stOperType.iFullSpeedStop THEN
					iRunStep:=iRunStep +3;
		ELSE
		 			iRunStep:=iRunStep +1;
 		END_IF
 2://参数传递
 		 iOldRunStep:=iRunStep;
 		 stPara.xStart:=TRUE;
		 IF   stPara.xBusy THEN
				 iRunStep:=iRunStep +1;
		 END_IF
 3://等待参数传递完成
 		 	iOldRunStep:=iRunStep;
 		 IF  stPara.xDone   THEN
				iRunStep:=iRunStep +1;
		 END_IF
 4://开始执行
 			iOldRunStep:=iRunStep;
	  IF 		 iOperType=stOperType.iPush OR
					 iOperType=stOperType.iPull  THEN
    				iRunStep:=10;
		ELSIF   iOperType=stOperType.iStop OR 
						iOperType=stOperType.iFullSpeedStop  THEN
    			  iRunStep:=20;
		ELSIF   iOperType=stOperType.iFullSpeedPull OR 
						iOperType=stOperType.iFullSpeedPush  THEN
		 				iRunStep:=30;
		ELSIF     iOperType=stOperType.iModulePush THEN
    				iRunStep:=40;
		ELSIF     iOperType=stOperType.iCalibAction THEN
    				iRunStep:=50;
		ELSIF  		iOperType=stOperType.iCalibInit THEN
		 				iRunStep:=60;
		ELSIF   		iOperType=stOperType.iAdjust THEN
		 				iRunStep:=70;
		END_IF	
 10://Pull/push
				iOldRunStep:=iRunStep;
				arwDataWriteRegs[1]:=1;//启动
				wQuantityWriteRegs:=1;
				wMBAddWriteRegs:=1011;
				xWriteRegs:=TRUE;
				IF  fbWriteRegs.bBusy THEN
						xWriteRegs:=FALSE;
						iRunStep:=iRunStep+1;
			 END_IF
 11://启动完成
			iOldRunStep:=iRunStep;
	  	IF  NOT 	fbWriteRegs.bBusy AND  NOT  	fbWriteRegs.bError THEN
	  	 				iRunStep:=iRunStep +1;
	  	 ELSIF   	fbWriteRegs.bError THEN
	  	 			iRunStep:=999;				
	  	 			eErrorID:=PumpError.FLT_RUN_ERROR;					
	  	 END_IF		
  12://等待运行结束
			iOldParaStep:=iParaStep;
			wMBAddReadRegs:=1011;
			wQuantityReadRegs:=1;
			xReadRegs:=TRUE;
			IF  fbReadRegs.bBusy THEN
			 	xReadRegs:=FALSE;
				iRunStep:=iRunStep+1;
			END_IF
	13://等待读取完成
			 	iOldParaStep:=iParaStep;
	  	  IF  NOT 	fbReadRegs.bBusy AND  NOT  	fbReadRegs.bError THEN
				 				 stReadPara.iRunning:=arwDataReadRegs[1];
	  		 				 iRunStep:=iRunStep+1;
	  		 ELSIF   	fbReadRegs.bError THEN
	  		 			iRunStep:=999;				
	  		 			eErrorID:=PumpError.FLT_READ_PARA;					
	  		 END_IF	
				 artDelay[1](IN:=FALSE);
	14://检查是否已经停止运行
				IF  stReadPara.iRunning =0 THEN
				 			iRunStep:=100;
				ELSE //再次读取
						artDelay[1](IN:= TRUE, PT:= T#100MS, Q=> , ET=> );
						IF  artDelay[1].Q  THEN
								 iRunStep:=12;
								 artDelay[1](IN:= FALSE);
						END_IF
				END_IF			 
	20://Stop
				 iOldRunStep:=iRunStep;
				 arwDataWriteRegs[1]:=0;//停止
				 arwDataWriteRegs[2]:=0;//全速停止
				 wQuantityWriteRegs:=2;
				 wMBAddWriteRegs:=1011;
				 xWriteRegs:=TRUE;
				 IF  fbWriteRegs.bBusy THEN
						 xWriteRegs:=FALSE;
						 iRunStep:=iRunStep+1;
				END_IF
	21://运行完成
			 iOldRunStep:=iRunStep;
			 IF  NOT 	fbWriteRegs.bBusy AND  NOT  	fbWriteRegs.bError THEN
							 iRunStep:=100;
				ELSIF   	fbWriteRegs.bError THEN
						 iRunStep:=999;				
						 eErrorID:=PumpError.FLT_RUN_ERROR;					
				END_IF				
	30://写入方向
				iOldParaStep:=iParaStep;
				MEMCPY(ADR(arwDataWriteRegs[1]),ADR(stLocalPara.iDirectionSet),SIZEOF (stLocalPara.iDirectionSet));
				wQuantityWriteRegs:=1;
				wMBAddWriteRegs:=1010;
				xWriteRegs:=TRUE;
				IF  fbWriteRegs.bBusy THEN
						xWriteRegs:=FALSE;
						iRunStep:=iRunStep+1;
			 END_IF
	 31://方向写入完成
			 iOldParaStep:=iParaStep;
			 IF  NOT 	fbWriteRegs.bBusy AND  NOT  	fbWriteRegs.bError THEN
							 iRunStep:=iRunStep +1;
				ELSIF   	fbWriteRegs.bError THEN
						 iRunStep:=999;				
						 eErrorID:=PumpError.FLT_SET_PARA;					
				END_IF		
	32://FullSpeed
				 iOldRunStep:=iRunStep;
				 arwDataWriteRegs[1]:=1;//全速启动
				 wQuantityWriteRegs:=1;
				 wMBAddWriteRegs:=1012;
				 xWriteRegs:=TRUE;
				 IF  fbWriteRegs.bBusy THEN
						 xWriteRegs:=FALSE;
						 iRunStep:=iRunStep+1;
				END_IF
	33://全速启动
			 iOldRunStep:=iRunStep;
			 IF  NOT 	fbWriteRegs.bBusy AND  NOT fbWriteRegs.bError THEN
							 iRunStep:=100;
				ELSIF   	fbWriteRegs.bError THEN
						 iRunStep:=999;				
						 eErrorID:=PumpError.FLT_RUN_ERROR;					
				END_IF	
	40://
			iCalibNum:=1;
			iRunStep:=iRunStep+1;
	41://Module Push
				 iOldRunStep:=iRunStep;
				 arwDataWriteRegs[1]:=1;//单元启动
				 wQuantityWriteRegs:=1;
				 wMBAddWriteRegs:=2003;
				 xWriteRegs:=TRUE;
				 IF  fbWriteRegs.bBusy THEN
						 xWriteRegs:=FALSE;
						 iRunStep:=iRunStep+1;
				END_IF
	42://单元启动注液
			 iOldRunStep:=iRunStep;
			 IF  NOT 	fbWriteRegs.bBusy AND  NOT fbWriteRegs.bError THEN
							 iRunStep:=iRunStep +1;
				ELSIF   	fbWriteRegs.bError THEN
						 iRunStep:=999;				
						 eErrorID:=PumpError.FLT_RUN_ERROR;					
				END_IF
	43://等待运行结束
			 iOldParaStep:=iParaStep;
			 wMBAddReadRegs:=2003;
			 wQuantityReadRegs:=1;
			 xReadRegs:=TRUE;
			 IF  fbReadRegs.bBusy THEN
				 xReadRegs:=FALSE;
				 iRunStep:=iRunStep+1;
			 END_IF
	 44://等待读取完成
				 iOldParaStep:=iParaStep;
				 IF  NOT 	fbReadRegs.bBusy AND  NOT  	fbReadRegs.bError THEN
									stReadPara.iRunning:=arwDataReadRegs[1];
									iRunStep:=iRunStep+1;
					ELSIF   	fbReadRegs.bError THEN
							 iRunStep:=999;				
							 eErrorID:=PumpError.FLT_READ_PARA;					
					END_IF	
					artDelay[1](IN:=FALSE);
	 45://检查是否已经停止运行
				 IF  stReadPara.iRunning =0 THEN
							 	iRunStep:=iRunStep +1;
				 ELSE //再次读取
						 artDelay[1](IN:= TRUE, PT:= T#100MS, Q=> , ET=> );
						 IF  artDelay[1].Q  THEN
									iRunStep:=12;
									artDelay[1](IN:= FALSE);
						 END_IF
				 END_IF		
		46://检查灌装次数
				iCalibNum:=iCalibNum +1 ;
				iRunStep:=iRunStep +1;
	  47://
				IF  iCalibNum > stLocalPara.iCycleNumber THEN
				 				iRunStep:=100;
				ELSE
								iRunStep:=iRunStep +1;		
				END_IF			 			 
		48://检查单元注液时间等待0.5
			 tModuleDelay(IN:=TRUE, PT:= T#1500MS, Q=> , ET=> );
			 IF	  	tModuleDelay.Q THEN
							 tModuleDelay(IN:=FALSE);	
							 iRunStep:=41;
			 END_IF	
			 
		50://写入实际液量	
					 MEMCPY(ADR(arwSetData[1]),ADR(stLocalPara.iModuleRealVolume),SIZEOF(stLocalPara.iModuleRealVolume) ); 
					 arwDataWriteRegs[1]:=arwSetData[2];
					 arwDataWriteRegs[2]:=arwSetData[1];
					 iRunStep:=iRunStep +1;
		
		51://开始写入
					 iOldRunStep:=iRunStep;
					 wQuantityWriteRegs:=2;
					 wMBAddWriteRegs:=2004;
					 xWriteRegs:=TRUE;
					 IF  fbWriteRegs.bBusy THEN
							 xWriteRegs:=FALSE;
							 iRunStep:=iRunStep+1;
					END_IF
		52://等待运行结束
				 iOldParaStep:=iParaStep;
				 wMBAddReadRegs:=1011;
				 wQuantityReadRegs:=1;
				 xReadRegs:=TRUE;
				 IF  fbReadRegs.bBusy THEN
					 xReadRegs:=FALSE;
					 iRunStep:=iRunStep+1;
				 END_IF
		 53://等待读取完成
					 iOldParaStep:=iParaStep;
					 IF  NOT 	fbReadRegs.bBusy AND  NOT  	fbReadRegs.bError THEN
										stReadPara.iRunning:=arwDataReadRegs[1];
										iRunStep:=iRunStep+1;
						ELSIF   	fbReadRegs.bError THEN
								 iRunStep:=999;				
								 eErrorID:=PumpError.FLT_READ_PARA;					
						END_IF	
						artDelay[1](IN:=FALSE);
		 54://检查是否已经停止运行
					 IF  stReadPara.iRunning =0 THEN
								 iRunStep:=100;
					 ELSE //再次读取
							 artDelay[1](IN:= TRUE, PT:= T#100MS, Q=> , ET=> );
							 IF  artDelay[1].Q  THEN
										iRunStep:=12;
										artDelay[1](IN:= FALSE);
							 END_IF
					 END_IF			 
		 60://初始化校准参数
					 stCalibInit.xStart :=TRUE;
					 iRunStep:=iRunStep +1;
		 61://等待
				 IF  stCalibInit.xBusy THEN
						 iRunStep:=iRunStep +1;
				 END_IF
		 62://完成
				 IF stCalibInit.xDone THEN
							 iRunStep:=100;
				 END_IF 
		 70://微调
					 stAdjust.xStart :=TRUE;
					 iRunStep:=iRunStep +1;
		 71://等待
				 IF  stAdjust.xBusy THEN
						 iRunStep:=iRunStep +1;
				 END_IF
		 72://完成
				 IF stAdjust.xDone THEN
							 iRunStep:=100;
				 END_IF 
	   100://等待S钟 
					artDelay[2](IN:=TRUE , PT:= T#1S, Q=> , ET=> );		 
					IF  artDelay[2].Q THEN
					     iRunStep:=iRunStep +1;
							 artDelay[2](IN:=FALSE);
					END_IF
		 101://运行结束
					xQBusy:=FALSE;
					xQDone:=TRUE;
					iRunStep:=0;
 END_CASE
 //防止程序二次执行
	IF  xQBusy THEN
		 		xStart:=FALSE;
  END_IF
END_ACTION

ACTION ACT_RunPara:
CASE iParaStep OF	
	0://开始
			IF   stPara.xStart THEN
			 		 stPara.xStart:=FALSE;
					 stPara.xBusy:=TRUE;
					 stPara.xDone:=FALSE;
					  iParaStep := iParaStep + 1;
			 END_IF
 	1://查流量设定的转速是否在0.1rpm-600rpm之间
			iOldParaStep:=iParaStep;
			IF 	stLocalPara.rRuntimeSet = 0  THEN 
					 eERRORID := PumpError.FLT_FLUVOLUM_TIME_PARA;		
					 iParaStep := 0;
		  ELSE
					rSetSpeed := stLocalPara.rFluVolumeSet * 60.0 / stRunPara.rSpeedRatio / stLocalPara.rRuntimeSet;
					IF rSetSpeed >= 0.001 AND  rSetSpeed <= 600 THEN
						iParaStep := iParaStep + 1;
					ELSE
						eERRORID := PumpError.FLT_FLUVOLUM_TIME_PARA;		
						iParaStep := 0;
			END_IF
		END_IF		
	2://读取液量（2word）、时间(2word)、间隔时间(2word)、灌装次数(word)、回吸角度(word)、运行方向(word)
			iOldParaStep:=iParaStep;
			wMBAddReadRegs:=1002;
			wQuantityReadRegs:=10;
			xReadRegs:=TRUE;
			IF  fbReadRegs.bBusy THEN
			 	xReadRegs:=FALSE;
				iParaStep:=iParaStep+1;
			END_IF
	3://等待读取完成
			 	iOldParaStep:=iParaStep;
	  	  IF  NOT 	fbReadRegs.bBusy AND  NOT  	fbReadRegs.bError THEN
				 				//液量
								stReadPara.rFluVolume:=M_Little_Endian(pInputData:=ADR(arwDataReadRegs[1]));
								//时间
								stReadPara.rRuntime:=M_Little_Endian(pInputData:=ADR(arwDataReadRegs[3]));
								
	  		 				 iParaStep:=iParaStep+1;
	  		 ELSIF   	fbReadRegs.bError THEN
	  		 			iParaStep:=999;				
	  		 			eErrorID:=PumpError.FLT_READ_PARA;					
	  		 END_IF	
	4://设定与显示进行比较
				iOldParaStep:=iParaStep;
				IF stLocalPara.rFluVolumeSet <> stReadPara.rFluVolume OR 
				 	 stLocalPara.rRuntimeSet <> stReadPara.rRuntime   THEN
					 iParaStep:=iParaStep + 1;	
				ELSE
					 iParaStep:=iParaStep+8;
				END_IF
	5://设定虚假时间
			 MEMCPY(ADR(arwSetData[1]),ADR(stLocalPara.rVirualTime),SIZEOF(stLocalPara.rVirualTime) ); 
			 arwDataWriteRegs[1]:=arwSetData[2];
			 arwDataWriteRegs[2]:=arwSetData[1];
			 iParaStep:=iParaStep +1;
	6://需要传送虚假的时间
			 iOldParaStep:=iParaStep;
			 wQuantityWriteRegs:=2;
			 wMBAddWriteRegs:=1004;
			 xWriteRegs:=TRUE;
			 IF  fbWriteRegs.bBusy THEN
					 xWriteRegs:=FALSE;
					 iParaStep:=iParaStep+1;
			END_IF	
	7://等待设定完成
				iOldParaStep:=iParaStep;
			 IF  NOT 	fbWriteRegs.bBusy AND  NOT  	fbWriteRegs.bError THEN
							  iParaStep:=iParaStep +1;
				ELSIF   	fbReadRegs.bError THEN
						 iParaStep:=999;				
						 eErrorID:=PumpError.FLT_SET_PARA;					
				END_IF				
  8://需要设定液量
			 iOldParaStep:=iParaStep;
			 MEMCPY(ADR(arwSetData[1]),ADR(stLocalPara.rFluVolumeSet),SIZEOF(stLocalPara.rFluVolumeSet) ); 
			 arwDataWriteRegs[1]:=arwSetData[2];
			 arwDataWriteRegs[2]:=arwSetData[1];
			 wQuantityWriteRegs:=2;
			 wMBAddWriteRegs:=1002;
			 xWriteRegs:=TRUE;
			 IF  fbWriteRegs.bBusy THEN
					 xWriteRegs:=FALSE;
					 iParaStep:=iParaStep+1;
			END_IF
	9://液量设定完成
			iOldParaStep:=iParaStep;
	  	IF  NOT 	fbWriteRegs.bBusy AND  NOT  	fbWriteRegs.bError THEN
	  	 				iParaStep:=iParaStep + 1;
	  	 ELSIF   	fbReadRegs.bError THEN
	  	 			iParaStep:=999;				
	  	 			eErrorID:=PumpError.FLT_SET_PARA;					
	  	 END_IF		
  10://设定运行时间
			 iOldParaStep:=iParaStep;
			 MEMCPY(ADR(arwSetData[1]),ADR(stLocalPara.rRuntimeSet),SIZEOF(stLocalPara.rRuntimeSet) ); 
			 arwDataWriteRegs[1]:=arwSetData[2];
			 arwDataWriteRegs[2]:=arwSetData[1];
			 wQuantityWriteRegs:=2;
			 wMBAddWriteRegs:=1004;
			 xWriteRegs:=TRUE;
			 IF  fbWriteRegs.bBusy THEN
					 xWriteRegs:=FALSE;
					 iParaStep:=iParaStep+1;
			END_IF
	11://等待时间设定完成
			iOldParaStep:=iParaStep;
	  	IF  NOT 	fbWriteRegs.bBusy AND  NOT  	fbWriteRegs.bError THEN
	  	 				iParaStep:=iParaStep + 1;
	  	 ELSIF   	fbReadRegs.bError THEN
	  	 			iParaStep:=999;				
	  	 			eErrorID:=PumpError.FLT_SET_PARA;					
	  	 END_IF		
	12://比较方向
				iOldParaStep:=iParaStep;
				stReadPara.iDirectionSet:=WORD_TO_INT(arwDataReadRegs[9]);
				IF stLocalPara.iDirectionSet<> stReadPara.iDirectionSet   THEN
										iParaStep:=iParaStep+1;	
				ELSE
										iParaStep:=iParaStep+3;	
				END_IF
	13://写入方向
			 iOldParaStep:=iParaStep;
			 MEMCPY(ADR(arwDataWriteRegs[1]),ADR(stLocalPara.iDirectionSet),SIZEOF (stLocalPara.iDirectionSet));
			 wQuantityWriteRegs:=1;
			 wMBAddWriteRegs:=1010;
			 xWriteRegs:=TRUE;
			 IF  fbWriteRegs.bBusy THEN
					 xWriteRegs:=FALSE;
					 iParaStep:=iParaStep+1;
			END_IF
  14://方向写入完成
			iOldParaStep:=iParaStep;
	  	IF  NOT 	fbWriteRegs.bBusy AND  NOT  	fbWriteRegs.bError THEN
	  	 				iParaStep:=iParaStep +1;
	  	 ELSIF   	fbReadRegs.bError THEN
	  	 			iParaStep:=999;				
	  	 			eErrorID:=PumpError.FLT_SET_PARA;					
	  	 END_IF		
	15://比较重复次数
				iOldParaStep:=iParaStep;
				//重复次数
				stReadPara.iCycleNumber:=WORD_TO_INT(arwDataReadRegs[7]);
				IF stLocalPara.iCycleNumber<> stReadPara.iCycleNumber   THEN
					 iParaStep:=iParaStep+1;	
				ELSE
					 iParaStep:=iParaStep+3;
				END_IF	
	16://写入重复次数
			 iOldParaStep:=iParaStep;
			 MEMCPY(ADR(arwDataWriteRegs[1]),ADR(stLocalPara.iCycleNumber),SIZEOF(stLocalPara.iCycleNumber));
			 wQuantityWriteRegs:=1;
			 wMBAddWriteRegs:=1008;
			 xWriteRegs:=TRUE;
			 IF  fbWriteRegs.bBusy THEN
					 xWriteRegs:=FALSE;
					 iParaStep:=iParaStep+1;
			END_IF
  17://重复次数写入完成
			iOldParaStep:=iParaStep;
	  	IF  NOT 	fbWriteRegs.bBusy AND  NOT  	fbWriteRegs.bError THEN
	  	 				iParaStep:=iParaStep +1;
	  	 ELSIF   	fbReadRegs.bError THEN
	  	 			iParaStep:=999;				
	  	 			eErrorID:=PumpError.FLT_SET_PARA;					
	  	 END_IF		
//////////////////////////待开放回吸角度/////////////////////////////////////////	 
	18://比较回吸角度
				iOldParaStep:=iParaStep;
				stReadPara.iBackAngle:=WORD_TO_INT(arwDataReadRegs[8]);
				IF stLocalPara.iBackAngle<> stReadPara.iBackAngle   THEN
					 iParaStep:=iParaStep+1;	
				ELSE
					 iParaStep:=iParaStep+3;
				END_IF	
	19://写入回吸角度
			 iOldParaStep:=iParaStep;
			 MEMCPY(ADR(arwDataWriteRegs[1]),ADR(stLocalPara.iBackAngle),SIZEOF(stLocalPara.iBackAngle));
			 wQuantityWriteRegs:=1;
			 wMBAddWriteRegs:=1009;
			 xWriteRegs:=TRUE;
			 IF  fbWriteRegs.bBusy THEN
					 xWriteRegs:=FALSE;
					 iParaStep:=iParaStep+1;
			END_IF
  20://写入回吸角度完成
			iOldParaStep:=iParaStep;
	  	IF  NOT 	fbWriteRegs.bBusy AND  NOT  	fbWriteRegs.bError THEN
	  	 				iParaStep:=iParaStep +1;
	  	 ELSIF   	fbReadRegs.bError THEN
	  	 			iParaStep:=999;				
	  	 			eErrorID:=PumpError.FLT_SET_PARA;					
	  	 END_IF				 
			 
	21://判断是否执行ModulePush
      IF   iOperType=stOperType.iModulePush THEN
						iParaStep:=iParaStep +1;
			ELSE
						iParaStep:=100;
			END_IF
	22://单元地址设定	
				 iOldParaStep:=iParaStep;
				 MEMCPY(ADR(arwDataWriteRegs[1]),ADR(stLocalPara.iModuleAdress),SIZEOF(stLocalPara.iModuleAdress));
				 wQuantityWriteRegs:=1;
				 wMBAddWriteRegs:=2000;
				 xWriteRegs:=TRUE;
				 IF  fbWriteRegs.bBusy THEN
						 xWriteRegs:=FALSE;
						 iParaStep:=iParaStep+1;
				END_IF
	23://单元地址设定完成
				iOldParaStep:=iParaStep;
				IF  NOT 	fbWriteRegs.bBusy AND  NOT  	fbWriteRegs.bError THEN
								iParaStep:=iParaStep +1;
				 ELSIF   	fbReadRegs.bError THEN
							iParaStep:=999;				
							eErrorID:=PumpError.FLT_SET_PARA;					
				 END_IF			
	24://写入回吸角度
				 iOldParaStep:=iParaStep;
				 MEMCPY(ADR(arwDataWriteRegs[1]),ADR(stLocalPara.iBackAngle),SIZEOF(stLocalPara.iBackAngle));
				 wQuantityWriteRegs:=1;
				 wMBAddWriteRegs:=1009;
				 xWriteRegs:=TRUE;
				 IF  fbWriteRegs.bBusy THEN
						 xWriteRegs:=FALSE;
						 iParaStep:=iParaStep+1;
				END_IF
	25://写入回吸角度完成
				iOldParaStep:=iParaStep;
				IF  NOT 	fbWriteRegs.bBusy AND  NOT  	fbWriteRegs.bError THEN
								iParaStep:=iParaStep +1;
				 ELSIF   	fbReadRegs.bError THEN
							iParaStep:=999;				
							eErrorID:=PumpError.FLT_SET_PARA;					
				 END_IF				 
	26://写入重复次数
			 iOldParaStep:=iParaStep;
			 MEMCPY(ADR(arwDataWriteRegs[1]),ADR(stLocalPara.iCycleNumber),SIZEOF(stLocalPara.iCycleNumber));
			 wQuantityWriteRegs:=1;
			 wMBAddWriteRegs:=1008;
			 xWriteRegs:=TRUE;
			 IF  fbWriteRegs.bBusy THEN
					 xWriteRegs:=FALSE;
					 iParaStep:=iParaStep+1;
			END_IF
  27://重复次数写入完成
			iOldParaStep:=iParaStep;
	  	IF  NOT 	fbWriteRegs.bBusy AND  NOT  	fbWriteRegs.bError THEN
	  	 				iParaStep:=100;
	  	 ELSIF   	fbReadRegs.bError THEN
	  	 			iParaStep:=999;				
	  	 			eErrorID:=PumpError.FLT_SET_PARA;					
	  	 END_IF				  

	//21://设定单元速度
	//		 iOldParaStep:=iParaStep;
	//		 MEMCPY(ADR(arwSetData[1]),ADR(stLocalPara.iModuleSpeed),SIZEOF(stLocalPara.iModuleSpeed) ); 
	//		 arwDataWriteRegs[1]:=arwSetData[2];
	//		 arwDataWriteRegs[2]:=arwSetData[1];
	//		 iParaStep:=iParaStep +1;
  //22://传送单元速度
	//		 iOldParaStep:=iParaStep;
	//		 wQuantityWriteRegs:=2;
	//		 wMBAddWriteRegs:=2001;
	//		 xWriteRegs:=TRUE;
	//		 IF  fbWriteRegs.bBusy THEN
	//				 xWriteRegs:=FALSE;
	//				 iParaStep:=iParaStep+1;
	//		END_IF	
	//23://等待设定完成
	//			iOldParaStep:=iParaStep;
	//		 IF  NOT 	fbWriteRegs.bBusy AND  NOT  	fbWriteRegs.bError THEN
	//						  iParaStep:=100;
	//			ELSIF   	fbReadRegs.bError THEN
	//					 iParaStep:=999;				
	//					 eErrorID:=PumpError.FLT_SET_PARA;					
	//			END_IF				
	100://参数写入完成
				iOperType:=stOperType.iWait;
				stPara.xBusy:=FALSE;
				stPara.xDone:=TRUE;
				iParaStep:=0;		
	ELSE
		;	
END_CASE
//防止程序二次执行
IF   stPara.xBusy THEN
		 stPara.xStart:=FALSE;
END_IF
END_ACTION

END_FUNCTION_BLOCK

// ---- POUs/003_FB/0015_Functions/001_Parallel/FC_ParallelFinished.TcPOU
FUNCTION FC_ParallelFinished : BOOL
(*return value=false: parallel process not finished *)
VAR_INPUT
	iIModuleNum:INT;(*module number*)
	iIRequestID:INT;(*source process ID*)
	iIExecuteID: INT; (*destination process ID*)
END_VAR
VAR
END_VAR

(*parallel process finish ,return value  true*)
IF asModuleSeqData[iIModuleNum].asSequenceData[iIExecuteID].xRunning AND asModuleSeqData[iIModuleNum].asSequenceData[iIExecuteID].xFinished THEN
	asModuleSeqData[iIModuleNum].asSequenceData[iIExecuteID].iRequestID:=-1;
	asModuleSeqData[iIModuleNum].asSequenceData[iIExecuteID].iJobNum:=0;
	asModuleSeqData[iIModuleNum].asSequenceData[iIExecuteID].xComplete:=TRUE;
	asModuleSeqData[iIModuleNum].asSequenceData[iIExecuteID].xFinished:=FALSE;
	asModuleSeqData[iIModuleNum].asSequenceData[iIExecuteID].xRequestSucceed:=FALSE;
	asModuleSeqData[iIModuleNum].asSequenceData[iIRequestID].aiParIDCreated[iIExecuteID]:=-1;
	asModuleSeqData[iIModuleNum].asSequenceData[iIRequestID].iNumOfParID:=asModuleSeqData[iIModuleNum].asSequenceData[iIRequestID].iNumOfParID-1;
	FC_ParallelFinished:=TRUE;
ELSE
	FC_ParallelFinished:=FALSE;
END_IF

END_FUNCTION

// ---- POUs/003_FB/0015_Functions/001_Parallel/FC_ParallelRequest.TcPOU
FUNCTION FC_ParallelRequest : BOOL
(*return value=false: parallel process is running *)
VAR_INPUT
	iIModuleNum:INT;(*module number*)
	iIRequestID:INT;(*source process ID*)
	iIExecuteID: INT; (*destination process ID*)
	iIJobNum:INT;(*program job num*)
END_VAR

VAR
END_VAR

(*process not running ,return value  true*)
IF asModuleSeqData[iIModuleNum].asSequenceData[iIExecuteID].iRequestID=-1 THEN
	asModuleSeqData[iIModuleNum].asSequenceData[iIExecuteID].iRequestID:=iIRequestID;
	asModuleSeqData[iIModuleNum].asSequenceData[iIExecuteID].iJobNum:=iIJobNum;
	asModuleSeqData[iIModuleNum].asSequenceData[iIExecuteID].xComplete:=FALSE;
	asModuleSeqData[iIModuleNum].asSequenceData[iIExecuteID].xRequestSucceed:=TRUE;
	asModuleSeqData[iIModuleNum].asSequenceData[iIRequestID].aiParIDCreated[iIExecuteID]:=1;
	asModuleSeqData[iIModuleNum].asSequenceData[iIRequestID].iNumOfParID:=asModuleSeqData[iIModuleNum].asSequenceData[iIRequestID].iNumOfParID+1;
	FC_ParallelRequest:=TRUE;
ELSE
	FC_ParallelRequest:=FALSE;
END_IF

END_FUNCTION

// ---- POUs/003_FB/19-AxisFB/FB_Axis_old.TcPOU
FUNCTION_BLOCK FB_Axis_old
VAR_INPUT
	xEStop								: BOOL;					//急停
	xKey									: BOOL;					//钥匙开关
	xSafety								: BOOL;					//安全防护
	xManualMode						: BOOL;					//手动模式
	xAutoMode							: BOOL;					//自动模式
	xAlarmReset						: BOOL;					//报警复位
	                  		
	xStop									: BOOL;					//轴停止
	xHalt									: BOOL;					//轴暂停
	xSv_not_power					: BOOL;					//轴断使能
	xNotPower       			: BOOL;					//轴断使能
	                  		
	xEnablePositive 			: BOOL:=TRUE;			//允许正转
	xEnableNegative				: BOOL:=TRUE;			//允许反转
	xRunILC								: BOOL:=TRUE;			//运行条件
	
	xPowerHmi							: BOOL;					//使能手动HMI
	xSetPosHmi						: BOOL;					//设置零点手动HMI
	xHomeHmi							: BOOL;					//原点搜索HMI
	xAlarmResetHmi				: BOOL;					//报警复位HMI
	xJogForwardHmi				: BOOL;					//Jog+HMI
	xJogBackwardsHmi			: BOOL;					//Jog-HMI
	xStopHmi					: BOOL;
	xJogForwardLimit  		: BOOL ;//JOG+极限
	xJogBackwardsLimit		: BOOL ;//JOG-极限
	
	xITarMoveHmi				:INT;//触摸屏选择 MMove Position
	xITarMoveButtonHmi			:BOOL;//触摸屏中目标位置按钮
	
	xPowerInit						: BOOL;					//使能初始化执行
	xHomeAuto							: BOOL;					//原点搜索自动执行
	xCalibrationCam				: BOOL;					//原点校准
	xJogForwardAuto				: BOOL;					//Jog+自动执行
	xJogBackwardsAuto			: BOOL;					//Jog-自动执行
	
	nMoveNum							: USINT:=6;				//轴绝对定位数量
	xMoveILC							: ARRAY[1..gc_uiAxisMoveNum] OF BOOL:=[gc_uiAxisMoveNum(TRUE)];//绝对定位动作条件
	xMoveHmi							: ARRAY[1..gc_uiAxisMoveNum] OF BOOL;//绝对定位手动Hmi
	xMoveAuto							: ARRAY[1..gc_uiAxisMoveNum] OF BOOL;//绝对定位自动执行
	
	rJogVelocity					: REAL;					//轴Jog速度
	rManualVelocity				: REAL;				//轴手动速度
	rAutoVelocity					: REAL;					//轴自动速度
	rMovePosition					: ARRAY[1..gc_uiAxisMoveNum] OF REAL;//绝对定位位置
	rMoveVelocity					: ARRAY[1..gc_uiAxisMoveNum] OF REAL;//绝对定位速度
	tInPosition						: ARRAY[1..gc_uiAxisMoveNum] OF TIME;//绝对到位延时
	rJogAcceleration      : REAL;                 //轴Jog加速度
	rJogDeceleration      : REAL;                 //轴Jog减速度
	rMoveAcceleration     : REAL;            //轴定位加速度                   	
	rMoveDeceleration     : REAL;           //轴定位减速度 
	rRelativeDistance			: REAL;					//相对定位位置
	rRelativeVelocity			: REAL;					//相对定位速度	
	rVelocityVel			    : REAL;					//连续运行速度
	rVelocityAcc			    : REAL;					//连续运行加速度
	rVelocityDec			    : REAL;					//连续运行减速度	
	
	iPosNumber						: INT;					//位置保存编号

	xRelativeILC        	: BOOL;                 //Relative条件
	xRelativeHmi			    : BOOL;					//相对定位手动Hmi
	xRelativeAuto			    : BOOL;					//相对定位自动执行
	
	xVelocityILC       		: BOOL;                 //Velocity条件
	xVelocityAuto			    : BOOL;					//连续运行启动
	xVelocityDirection		: BOOL;                 //连续运行方向  

	
	xModulo								: BOOL;					//模长内定位启动
	rModuloPosition				: REAL;					//模长内定位位置
	rModuloVelocity				: REAL;					//模长内定位速度
	nModuloDirection			: INT := (MC_Direction.MC_Positive_Direction);//模长定位方向
	tMoveTimeout					: TIME:=T#10S;			//定位超时
	wManualTip						: BYTE;					//手动提示字节,用于外部触发
	{attribute 'hide'}
	iHomingMode     : INT ; //回原模式输入
	{attribute 'hide'}
	xIsLinearMode : BOOL := TRUE;//默认都是线性模式	
END_VAR

VAR_OUTPUT
	xPowerOn							: BOOL;					//使能On
	xSetPosFinish					: BOOL;					//设置零点完成
	xReady								: BOOL;					//准备好
	xMoveDone							: ARRAY[1..gc_uiAxisMoveNum] OF BOOL;//绝对定位完成
	xMoveInPos						: ARRAY[1..gc_uiAxisMoveNum] OF BOOL;//绝对定位到位
	xMoveTimeout					: BOOL;					//定位超时报警
	xNotPowerOn						: BOOL;					//使能未On提示
	
	xError								: BOOL;					//错误
	xbusy									: BOOL;
	nErrorID							: UDINT;				//错误ID
	nErrorCode						: UDINT;				//错误代码
	
	rSetTorque						: REAL;					//设定转矩
	rSetPos								: REAL;					//设定位置
	rModuloSetPos					: REAL;					//模长内定位设定位置
	rModuloSetTurns				: REAL;					//模长内定位设定匝数
	rTargetPos						: REAL;					//目标位置
	
	rActTorque						: REAL;					//当前转矩
	rActPos								: REAL;					//当前位置
	rActVelo							: REAL;					//当前速度
	rModuloActPos					: REAL;					//模长内定位当前位置
	rModuloActTurns				: REAL;					//模长内定位当前匝数
	rPosDiff							: REAL;					//跟随误差

	xRelativeDone1				: BOOL;					//相对定位完成标志	
	xRelativeDone					: BOOL;					//相对定位完成
	xRelativeBusy					: BOOL;					//相对定位Busy
	xRelativeError				: BOOL;					//相对定位错误
	udiRelativeErrorID		: UDINT;				//相对定位错误ID
	
	xVelocityInVel				: BOOL;					//连续运行速度到达
	xVelocityBusy					: BOOL;					//连续运行Busy
	xVelocityError				: BOOL;					//连续运行错误
	udiVelocityErrorID		: UDINT;				//连续运行错误ID	
	
	
	xQTarPosition			:REAL;//触摸屏中显示在目标位置中
	xQTarVelocity			:REAL;//触摸屏中显示在目标速度中
	{attribute 'hide'}
	NcToPlc								: NCTOPLC_AXIS_REF;		//轴NcToPlc结构体
	{attribute 'hide'}
	Status								: ST_AxisStatus;		//轴状态结构体
END_VAR

VAR_IN_OUT
	{attribute 'hide'}
	Axis									: AXIS_REF;				//轴
END_VAR

VAR
	{attribute 'hide'}
	rtPowerHmi						: R_TRIG;				//使能手动HMI上升沿
	{attribute 'hide'}
	rtSetPosHmi						: R_TRIG;				//设置零点手动HMI上升沿
	{attribute 'hide'}
	xPowerManual					: BOOL;					//使能手动执行
	{attribute 'hide'}
	xPowerAuto						: BOOL;					//使能自动执行
	{attribute 'hide'}
	xPowerEnable					: BOOL;					//使能Enable
	{attribute 'hide'}
	rtPowerOn							: R_TRIG;				//使能上升沿
	{attribute 'hide'}
	rtPowerOff						: R_TRIG;				//使能下降沿
	{attribute 'hide'}
	xRunable							: BOOL;					//可运行
	{attribute 'hide'}
	xHomeManual						: BOOL;					//回原点手动执行
	{attribute 'hide'}
	xHomeExecute					: BOOL;					//回原点触发
	{attribute 'hide'}
	xSetPosExecute				: BOOL;					//设置零点触发
	{attribute 'hide'}
	xResetExecute					: BOOL;					//复位
	{attribute 'hide'}
	xJogForwardManual			: BOOL;					//Jog+手动执行
	{attribute 'hide'}
	xJogBackwardsManual		: BOOL;					//Jog-自动执行
	{attribute 'hide'}
	xJogForward						: BOOL;					//Jog+
	{attribute 'hide'}
	xJogBackwards					: BOOL;					//Jog-
	{attribute 'hide'}
	xMoveManual						: ARRAY[1..gc_uiAxisMoveNum] OF BOOL;//绝对定位手动执行
	{attribute 'hide'}
	xMoveExecute					: ARRAY[1..gc_uiAxisMoveNum] OF BOOL;//绝对定位启动使能
	{attribute 'hide'}
	xRelativeExecute			: BOOL;					//相对定位启动
	{attribute 'hide'}
	xModuloExecute				: BOOL;					//模长内定位启动
	{attribute 'hide'}
	xVelocityExecute			: BOOL;					//相对定位启动
	{attribute 'hide'}
	xVelocityAble			    : BOOL;					//相对定位使能
	{attribute 'hide'}
	rVelocity							:	REAL;					//定位速度
	{attribute 'hide'}
	nIndex 								:	INT;//索引
	{attribute 'hide'}
	tonInPosition					: ARRAY[1..gc_uiAxisMoveNum] OF TON;//绝对定位到位计时
	{attribute 'hide'}
	tonMoveTimeout				: ARRAY[1..gc_uiAxisMoveNum] OF TON;//绝对定位超时
	{attribute 'hide'}
	nIndexMove						: UINT;					//绝对定位索引
	{attribute 'hide'}
	xHaltExecute					: BOOL;					//轴暂停
	{attribute 'hide'}
	xStopExecute					: BOOL;					//轴停止
	{attribute 'hide'}
	fbReadStatus					: MC_ReadStatus;		//读取状态功能块
	{attribute 'hide'}
	fbPower								: MC_Power;				//使能功能块
	{attribute 'hide'}
	fbJog									: MC_Jog;				//Jog功能块
	{attribute 'hide'}
	fbHome								: MC_Home;				//原点搜索功能块
	{attribute 'hide'}
	fbMove								: ARRAY[1..gc_uiAxisMoveNum] OF MC_MoveAbsolute;//绝对定位功能块
	{attribute 'hide'}
	fbRelative					: MC_MoveRelative;		//相对定位功能块
	{attribute 'hide'}
	fbVelocity						: MC_MoveVelocity;	    //轴速度运行功能块
	{attribute 'hide'}
	fbModulo							: MC_MoveModulo;		//模长内定位
	{attribute 'hide'}
	fbReset								: MC_Reset;				//错误复位功能块
	{attribute 'hide'}
	fbHalt								: MC_Halt;				//轴暂停功能块
	{attribute 'hide'}
	fbStop								: MC_Stop;				//轴停止功能块
	{attribute 'hide'}
	fbSetPos							: MC_SetPosition;		//设置原点位置
END_VAR

ACT_ReadStatus();
ACT_Power();
ACT_Jog();
ACT_Home();
IF xIsLinearMode//判断是是否是线性模式
THEN
	ACT_Move();//线性模式运动调用
ELSE
	ACT_Modulo();//模值模式调用
END_IF

ACT_Relative();
ACT_InPos();
ACT_Timeout();
ACT_Tip();
ACT_Reset();
ACT_Halt();
ACT_Stop();
ACT_Velocity();

xPowerHmi:=FALSE;
xHomeHmi:=FALSE;
xAlarmResetHmi:=FALSE;
xPowerInit:=FALSE;
xHomeAuto:=FALSE;
//xJogForwardAuto:=FALSE;
//xJogBackwardsAuto:=FALSE;
xModulo:=FALSE;
xRelativeAuto:=FALSE;

FOR nIndex:=1 TO gc_uiAxisMoveNum DO
	//xMoveHmi[nIndex]:=FALSE;
	xMoveAuto[nIndex]:=FALSE;
END_FOR

ACTION ACT_Halt:

xHaltExecute:=xHalt;
fbHalt(
	Axis:=Axis,
	Execute:=xHaltExecute,
	Deceleration:=,
	Jerk:=,
	BufferMode:=,
	Options:=,
	Done=>,
	Busy=>,
	Active=>,
	CommandAborted=>,
	Error=>,
	ErrorID=>
);
END_ACTION

ACTION ACT_Home:

xHomeManual:=xHomeHmi
	AND xManualMode;
xHomeExecute:=xRunable
	AND (xHomeManual
		OR xHomeAuto
	);
fbHome(
	Axis:=Axis,
	Execute:=xHomeExecute,
	Position:=0,
	HomingMode:=iHomingMode,
	BufferMode:=,
	Options:=,
	bCalibrationCam:=xCalibrationCam,
	Done=>,
	Busy=>,
	Active=>,
	CommandAborted=>,
	Error=>,
	ErrorID=>
);
END_ACTION

ACTION ACT_InPos:

(*FOR nIndexMove:=1 TO nMoveActualNum DO
	tonInPosition[nIndexMove](
		IN:=bReady
			AND NOT Axis.Status.Moving
			AND Axis.Status.NotMoving
			AND Axis.Status.InPositionArea
			AND Axis.Status.InTargetPosition
			AND Axis.NcToPlc.SetPos=REAL_TO_LREAL(rMovePosition[nIndexMove])
			AND Axis.NcToPlc.TargetPos=REAL_TO_LREAL(rMovePosition[nIndexMove]),
		PT:=tInPosition[nIndexMove],
		Q=>bInPosition[nIndexMove],
		ET=>
	);
END_FOR*)
//检测运行是否到位
IF xIsLinearMode THEN //线性定位
	FOR nIndexMove:=1 TO gc_uiAxisMoveNum DO
		tonInPosition[nIndexMove](
			IN:=xReady
			 AND NOT Axis.Status.Moving
			 AND Axis.Status.NotMoving
			//   AND Axis.Status.InPositionArea
			//   AND Axis.Status.InTargetPosition
			//   AND Axis.NcToPlc.SetPos=REAL_TO_LREAL(rMovePosition[nIndexMove])
			//   AND Axis.NcToPlc.TargetPos=REAL_TO_LREAL(rMovePosition[nIndexMove]),
			 AND Axis.NcToPlc.ActPos >= REAL_TO_LREAL(rMovePosition[nIndexMove] - 0.2)
			 AND Axis.NcToPlc.ActPos <= REAL_TO_LREAL(rMovePosition[nIndexMove] + 0.2),
			PT:=tInPosition[nIndexMove],
			Q=>xMoveInPos[nIndexMove],
			ET=>);
	END_FOR
ELSE//模值定位
		FOR nIndexMove:=1 TO gc_uiAxisMoveNum DO
		tonInPosition[nIndexMove](
			IN:=xReady
			 AND NOT Axis.Status.Moving
			 AND Axis.Status.NotMoving
			//   AND Axis.Status.InPositionArea
			//   AND Axis.Status.InTargetPosition
			//   AND Axis.NcToPlc.SetPos=REAL_TO_LREAL(rMovePosition[nIndexMove])
			//   AND Axis.NcToPlc.TargetPos=REAL_TO_LREAL(rMovePosition[nIndexMove]),
			 AND Axis.NcToPlc.ModuloActPos >= REAL_TO_LREAL(rMovePosition[nIndexMove] - 0.2)
			 AND Axis.NcToPlc.ModuloActPos <= REAL_TO_LREAL(rMovePosition[nIndexMove] + 0.2),
			PT:=tInPosition[nIndexMove],
			Q=>xMoveInPos[nIndexMove],
			ET=>);
	END_FOR
END_IF
END_ACTION

ACTION ACT_Jog:

xJogForwardManual:=xJogForwardHmi
	AND xManualMode;
xJogBackwardsManual:=xJogBackwardsHmi
	AND xManualMode;
xJogForward:=xRunable
	AND NOT xJogBackwards
	AND NOT xJogForwardLimit
	AND (xJogForwardManual
		OR xJogForwardAuto
	);
xJogBackwards:=xRunable
	AND NOT xJogForward
	AND NOT xJogBackwardsLimit
	AND (xJogBackwardsManual
		OR xJogBackwardsAuto
	);
fbJog(
	Axis:=Axis,
	JogForward:=xJogForward,
	JogBackwards:=xJogBackwards,
	Mode:=MC_JOGMODE_CONTINOUS,
	Position:=0,
	Velocity:=REAL_TO_LREAL(rJogVelocity),
	Acceleration:=(*REAL_TO_LREAL(rJogAcceleration)*),
	Deceleration:=(*REAL_TO_LREAL(rJogDeceleration)*),
	Jerk:=,
	Done=>,
	Busy=>,
	Active=>,
	CommandAborted=>,
	Error=>,
	ErrorID=>
);
END_ACTION

ACTION ACT_Modulo:
FOR nIndexMove:=1 TO gc_uiAxisMoveNum DO
	IF xAutoMode THEN
		IF rMoveVelocity[nIndexMove]>0 
		THEN
			rVelocity:=rMoveVelocity[nIndexMove];
		ELSE
			rVelocity:=rAutoVelocity;
		END_IF
	ELSE
		rVelocity:=rManualVelocity;
	END_IF	
	
	xMoveManual[nIndexMove]:=xMoveHmi[nIndexMove] AND xMoveILC[nIndexMove]
													AND xManualMode;
	xMoveExecute[nIndexMove]:=xRunable
														AND xMoveILC[nIndexMove]
														AND (xMoveManual[nIndexMove]
														OR xMoveAuto[nIndexMove]);
	fbModulo(
		Axis:=Axis,
		Execute:=xMoveExecute[nIndexMove],
		Position:=REAL_TO_LREAL(rMovePosition[nIndexMove]),
		Velocity:=REAL_TO_LREAL(rVelocity),
		Acceleration:=REAL_TO_LREAL(rMoveAcceleration),
		Deceleration:=REAL_TO_LREAL(rMoveDeceleration),
		Direction:=nModuloDirection,
		BufferMode:=,
		Options:=,
		Done=>,
		Busy=>,
		Active=>,
		CommandAborted=>,
		Error=>,
		ErrorID=>
	);
END_FOR
END_ACTION

ACTION ACT_Move:

FOR nIndexMove:=1 TO gc_uiAxisMoveNum DO
	IF xAutoMode THEN
		IF rMoveVelocity[nIndexMove]>0 
		THEN
			rVelocity:=rMoveVelocity[nIndexMove];
		ELSE
			rVelocity:=rAutoVelocity;
		END_IF
	ELSE
		rVelocity:=rManualVelocity;
	END_IF	
	
	xMoveManual[nIndexMove]:=xMoveHmi[nIndexMove] AND xMoveILC[nIndexMove]
													AND xManualMode;
	xMoveExecute[nIndexMove]:=xRunable AND xMoveILC[nIndexMove]
										AND (xMoveManual[nIndexMove]
										OR xMoveAuto[nIndexMove]);
	fbMove[nIndexMove](
		Axis:=Axis,
		Execute:=xMoveExecute[nIndexMove],
		Position:=REAL_TO_LREAL(rMovePosition[nIndexMove]),
		Velocity:=REAL_TO_LREAL(rVelocity),
		Acceleration:=REAL_TO_LREAL(rMoveAcceleration),
		Deceleration:=REAL_TO_LREAL(rMoveDeceleration),
		Jerk:=,
		BufferMode:=MC_Aborting,
		Options:=,
		Done=>xMoveDone[nIndexMove],
		Busy=>,
		Active=>,
		CommandAborted=>,
		Error=>,
		ErrorID=>
	);
END_FOR
(**********************************触摸屏中选择伺服参数************************************)
xMoveExecute[xITarMoveHmi]:=xITarMoveButtonHmi;
xQTarPosition			:=rMovePosition[xITarMoveHmi];
xQTarVelocity			:=rManualVelocity;
END_ACTION

ACTION ACT_Power:

rtPowerHmi(
	CLK:=xPowerHmi,
	Q=>
);
IF xEStop AND xSafety THEN
	IF rtPowerHmi.Q
		AND xKey
		AND xSafety
		AND xManualMode
	THEN
		xPowerManual:=NOT xPowerManual;
	END_IF
	IF xPowerInit THEN
		xNotPower:=FALSE;
		xPowerManual:=FALSE;
		xPowerAuto:=TRUE;
	END_IF
ELSE
	xPowerManual:=FALSE;
	xPowerAuto:=FALSE;
END_IF
xPowerEnable:=NOT Axis.Status.Error
						AND (xPowerManual XOR xPowerAuto);
fbPower(
	Axis:=Axis,
	Enable:=xPowerEnable AND NOT xSv_not_power AND NOT xNotPower,
	Enable_Positive:=xEnablePositive,
	Enable_Negative:=xEnableNegative,
	Override:=100,
	BufferMode:=,
	Options:=,
	Status=>xPowerOn,
	Busy=>,
	Active=>,
	Error=>,
	ErrorID=>
);
//xPowerOn := Axis.NcToPlc.StateDWord.1;
//Axis.Status;
//AXIS.NcToPlc.StateDWord;
//AXIS.NcToPlc.StateDWord2;
//AXIS.NcToPlc.StateDWord3;
uiStatusCopy[2].1;
uiStatusCopy[2];
xReady:=xPowerOn
	AND NOT Axis.Status.Error
	AND Axis.Status.Operational;
xRunable:=xEStop
	AND xKey
	AND xSafety
	AND xReady
	AND xRunILC;
END_ACTION

ACTION ACT_ReadStatus:

fbReadStatus(
	Axis:=Axis,
	Enable:=TRUE,
	Valid=>,
	Busy=>,
	Error=>,
	ErrorID=>,
	ErrorStop=>,
	Disabled=>,
	Stopping=>,
	StandStill=>,
	DiscreteMotion=>,
	ContinuousMotion=>,
	SynchronizedMotion=>,
	Homing=>,
	ConstantVelocity=>,
	Accelerating=>,
	Decelerating=>,
	Status=>
);

xError					:=Axis.Status.Error;
nErrorID				:=Axis.Status.ErrorID;
xbusy					:=Axis.Status.Moving;
nErrorCode				:=Axis.NcToPlc.ErrorCode;


rSetTorque				:=LREAL_TO_REAL(Axis.NcToPlc.SetTorque);
rSetPos					:=LREAL_TO_REAL(Axis.NcToPlc.SetPos);
rModuloSetPos			:=LREAL_TO_REAL(Axis.NcToPlc.ModuloSetPos);
rModuloSetTurns			:=LREAL_TO_REAL(Axis.NcToPlc.ModuloSetTurns);
rTargetPos				:=LREAL_TO_REAL(Axis.NcToPlc.TargetPos);

rActTorque				:=LREAL_TO_REAL(Axis.NcToPlc.ActTorque);
IF xIsLinearMode//判断是是否是线性模式(不同模式读取的数据源不同)
THEN
	rActPos					:=LREAL_TO_REAL(Axis.NcToPlc.ActPos);
ELSE
	rActPos			    :=LREAL_TO_REAL(Axis.NcToPlc.ModuloActPos);
END_IF
rActVelo				:=LREAL_TO_REAL(Axis.NcToPlc.ActVelo);

rPosDiff				:=LREAL_TO_REAL(Axis.NcToPlc.PosDiff);

NcToPlc					:=Axis.NcToPlc;
Status					:=Axis.Status;
END_ACTION

ACTION ACT_Relative:
IF xAutoMode THEN
	IF rRelativeVelocity>0 THEN
		rVelocity:=rRelativeVelocity;
	ELSE
		rVelocity:=rAutoVelocity;
	END_IF
ELSE
	rVelocity:=rManualVelocity;
END_IF
xRelativeExecute:=xRunable
		AND ((xRelativeHmi AND xManualMode) OR xRelativeAuto (*AND xAutoMode*)) AND xRelativeILC;

fbRelative(
	Axis:=Axis,  
	Execute:= xRelativeExecute, 
	Distance:= REAL_TO_LREAL(rRelativeDistance), 
	Velocity:= REAL_TO_LREAL(rVelocity), 
	Acceleration:= rMoveAcceleration, 
	Deceleration:= rMoveDeceleration, 
	Jerk:= , 
	Done=> xRelativeDone, 
	Busy=> xRelativeBusy, 
	CommandAborted=> , 
	Error=> xRelativeError, 
	ErrorID=> udiRelativeErrorID);
	
IF xRelativeDone=TRUE THEN
	xRelativeDone1:=TRUE;
ELSIF xRelativeBusy=TRUE THEN
	xRelativeDone1:=FALSE;	
END_IF//
END_ACTION

ACTION ACT_Reset:
xResetExecute:=xAlarmReset
	OR xAlarmResetHmi;
	
fbReset(
	Axis:=Axis,
	Execute:=xResetExecute AND ( Axis.Status.Error OR NOT xPowerOn) ,
	Done=>,
	Busy=>,
	Error=>,
	ErrorID=>
);
END_ACTION

ACTION ACT_Stop:

xStopExecute:=xStop OR (xStopHmi AND xManualMode);
fbStop(
	Axis:=Axis,
	Execute:=xStopExecute,
	Deceleration:=,
	Jerk:=,
	Options:=,
	Done=>,
	Busy=>,
	Active=>,
	CommandAborted=>,
	Error=>,
	ErrorID=>
);
END_ACTION

ACTION ACT_Timeout:

IF xResetExecute THEN
	xMoveTimeout:=FALSE;
END_IF

IF NOT xMoveTimeout THEN
	FOR nIndexMove:=1 TO gc_uiAxisMoveNum DO
		tonMoveTimeout[nIndexMove](
			IN:=xMoveAuto[nIndexMove],
			PT:=tMoveTimeout,
			Q=>, ET=>
		);
		IF tonMoveTimeout[nIndexMove].Q THEN
			xMoveTimeout:=TRUE;
			EXIT;
		END_IF
	END_FOR
END_IF
END_ACTION

ACTION ACT_Tip:

IF xResetExecute THEN
	wManualTip:=0;
	xNotPowerOn:=FALSE;
END_IF

IF NOT (xPowerManual XOR xPowerAuto) 
	AND xAutoMode
	AND NOT Axis.Status.Error
THEN
	xNotPowerOn:=TRUE;
END_IF
END_ACTION

ACTION ACT_Velocity:
IF xAutoMode THEN
	IF rVelocityVel>0 THEN
		fbVelocity.Velocity:=rVelocityVel;
	ELSE
		fbVelocity.Velocity:=rAutoVelocity;
	END_IF
ELSE
	fbVelocity.Velocity:=rManualVelocity;
END_IF
xVelocityExecute:=xRunable AND xVelocityAuto AND xVelocityILC;

fbVelocity(
	Axis:=Axis , 
	Execute:=xVelocityExecute AND xVelocityAble , 
	Velocity:= , 
	Acceleration:=rVelocityAcc , 
	Deceleration:=rVelocityDec , 
	Jerk:= , 
	Direction:= , 
	InVelocity=>xVelocityInVel , 
	Busy=>xVelocityBusy , 
	CommandAborted=> , 
	Error=>xVelocityError , 
	ErrorID=>udiVelocityErrorID );
	
xVelocityAble:= NOT xVelocityAble;
END_ACTION

END_FUNCTION_BLOCK

// ---- POUs/003_FB/43_implicit checks/CheckBounds.TcPOU
// 隐含生成代码：不要编辑
FUNCTION CheckBounds : DINT
VAR_INPUT
	index, lower, upper: DINT;
END_VAR

// 隐含生成代码：这里只是对代码实现的建议
{noflow}
IF  index < lower THEN
	CheckBounds := lower;
ELSIF  index > upper THEN
	CheckBounds := upper;
ELSE  
	CheckBounds := index;
END_IF
{flow}

END_FUNCTION

// ---- POUs/003_FB/43_implicit checks/CheckDivDInt.TcPOU
// 隐含生成代码：不要编辑
FUNCTION CheckDivDInt : DINT
VAR_INPUT
	divisor:DINT;
END_VAR

// 隐含生成代码：这里只是对代码实现的建议
{noflow}
IF divisor = 0 THEN
	CheckDivDInt:=1;
ELSE
	CheckDivDInt:=divisor;
END_IF;
{flow}

END_FUNCTION

// ---- POUs/003_FB/43_implicit checks/CheckDivLInt.TcPOU
// 隐含生成代码：不要编辑
FUNCTION CheckDivLInt : LINT
VAR_INPUT
	divisor:LINT;
END_VAR

// 隐含生成代码：这里只是对代码实现的建议
{noflow}
IF divisor = 0 THEN
	CheckDivLInt:=1;
ELSE
	CheckDivLInt:=divisor;
END_IF;
{flow}

END_FUNCTION

// ---- POUs/003_FB/43_implicit checks/CheckDivLReal.TcPOU
// 隐含生成代码：不要编辑
FUNCTION CheckDivLReal : LREAL
VAR_INPUT
	divisor:LREAL;
END_VAR

// 隐含生成代码：这里只是对代码实现的建议
{noflow}
IF divisor = 0 THEN
	CheckDivLReal:=1;
ELSE
	CheckDivLReal:=divisor;
END_IF;
{flow}

END_FUNCTION

// ---- POUs/003_FB/43_implicit checks/CheckDivReal.TcPOU
// 隐含生成代码：不要编辑
FUNCTION CheckDivReal : REAL
VAR_INPUT
	divisor:REAL;
END_VAR

// 隐含生成代码：这里只是对代码实现的建议
{noflow}
IF divisor = 0 THEN
	CheckDivReal:=1;
ELSE
	CheckDivReal:=divisor;
END_IF;
{flow}

END_FUNCTION

// ---- POUs/003_FB/43_implicit checks/CheckLRangeSigned.TcPOU
// 隐含生成代码：不要编辑
FUNCTION CheckLRangeSigned : LINT
VAR_INPUT
	value, lower, upper: LINT;
END_VAR

// 隐含生成代码：这里只是对代码实现的建议
{noflow}
IF (value < lower) THEN
	CheckLRangeSigned := lower;
ELSIF(value > upper) THEN
	CheckLRangeSigned := upper;
ELSE
	CheckLRangeSigned := value;
END_IF

{flow}

END_FUNCTION

// ---- POUs/003_FB/43_implicit checks/CheckLRangeUnsigned.TcPOU
// 隐含生成代码：不要编辑
FUNCTION CheckLRangeUnsigned : ULINT
VAR_INPUT
	value, lower, upper: ULINT;
END_VAR

// 隐含生成代码：这里只是对代码实现的建议
{noflow}
IF (value < lower) THEN
	CheckLRangeUnsigned := lower;
ELSIF(value > upper) THEN
	CheckLRangeUnsigned := upper;
ELSE
	CheckLRangeUnsigned := value;
END_IF
{flow}

END_FUNCTION

// ---- POUs/003_FB/43_implicit checks/CheckPointer.TcPOU
// 隐含生成代码：不要编辑
FUNCTION CheckPointer : POINTER TO BYTE
VAR_INPUT 
	ptToTest : POINTER TO BYTE; // 指针的目标地址
	iSize : DINT;		        // 指针指向的类型大小。（例如：POINTER TO ARRAY [0..9] OF INT为20）
	iGran : DINT;		        // 指针访问的粒度，即指针指向的类型中最大的非结构数据类型的大小。（例如：POINTER TO ARRAY [0..9] OF INT为2）
	bWrite: BOOL;		        // 指示读或写权限。TRUE=写权限。
END_VAR

